(* OpticalPowermeterConfigs *) 
IF Config.OpticalPowermeterConfigs.PM101OpticalPowermeterConfigHs.IsEnabled THEN
	PM101OpticalPowermeterHs.FB_init(FALSE, FALSE, Config := Config.OpticalPowermeterConfigs.PM101OpticalPowermeterConfigHs, 
												   PolarisationConfig := CalibrateConfig.HSPowermeter.PolarisationConfig, 
												   RFactorSettings := CalibrateConfig.HSPowermeter.RFactorSettings,
												   ResponsivityConfig := CalibrateConfig.HSPowermeter.ResponsivityConfig);		
END_IF
IF Config.OpticalPowermeterConfigs.PM101OpticalPowermeterConfigHt.IsEnabled THEN
	PM101OpticalPowermeterHt.FB_init(FALSE, FALSE, Config := Config.OpticalPowermeterConfigs.PM101OpticalPowermeterConfigHt, 
												   PolarisationConfig := CalibrateConfig.HTPowermeter.PolarisationConfig,
												   RFactorSettings := CalibrateConfig.HTPowermeter.RFactorSettings,
												   ResponsivityConfig := CalibrateConfig.HTPowermeter.ResponsivityConfig);
END_IF

(* DistanceSensorConfigs *) 
IF Config.DistanceSensorConfigs.MicroEpsilonDistanceSensorConfig.IsEnabled THEN
	MicroEpsilonDistanceSensor.FB_init(FALSE, FALSE, Config := Config.DistanceSensorConfigs.MicroEpsilonDistanceSensorConfig);	
END_IF

(* MppcConfigs *) 
IF Config.MppcConfigs.C13336MppcConfigWide.IsEnabled THEN
	C13336MppcWide.FB_init(FALSE, FALSE, Config := Config.MppcConfigs.C13336MppcConfigWide);	
END_IF
IF Config.MppcConfigs.C13336MppcConfigNarrow.IsEnabled THEN
	C13336MppcNarrow.FB_init(FALSE, FALSE, Config := Config.MppcConfigs.C13336MppcConfigNarrow);	
END_IF

(* ShutterConfigs *) 
IF Config.ShutterConfigs.Ed12dssShutterConfig.IsEnabled THEN
	Ed12dssShutter.FB_init(FALSE, FALSE, Config := Config.ShutterConfigs.Ed12dssShutterConfig);	
ELSIF Config.ShutterConfigs.SH10PILShutterConfig.IsEnabled THEN
	Sh10pilShutter.FB_init(FALSE, FALSE, Config := Config.ShutterConfigs.SH10PILShutterConfig);	
END_IF

IF Config.IsEnabled THEN
	_logger.Information('Lightspeed devices initialization ended...');
END_IF
END_METHOD

METHOD OpenCloseCycling : BOOL
VAR_INPUT
	Execute : BOOL;
	Count : UINT;
END_VAR
VAR 
END_VAR
IF Execute THEN
	(* timer pour l'enchainement des open/close *)
	(* WaitingTimer.in := TRUE;
	WaitingTimer.PT := T#4S;*)
	WaitingTimer (IN :=TRUE , PT := T#5S,Q=>, ET=> );
	
	(* WaitingTimer.Q is TRUE, PT seconds after IN had a rising edge *)
	IF WaitingTimer.Q THEN
		(* RAZ du timer *)
		WaitingTimer (IN := FALSE);
		(* coupe le motor ON par securité*)
		Chamber.IoLightspeed.OutputDoorslitMotorOn := FALSE;
		(* MAJ du compteur*)
		OpenCloseCyclingCount := Count;
		(* porte ouverte => on demande la fermeture*)
		IF (_CyclingCounterReachSetpoint) THEN
			(* arret du cycling et re init des variables*)
			Chamber.IoLightspeed.OutputDoorslitMotorOn := FALSE;
			_startCycling := FALSE;
			_CyclingCounterReachSetpoint := FALSE;
			_ActivateCyclingMotorOpen := FALSE;
			OpenCloseCycling := FALSE;
			OpenCloseCurrentCounterValue := 0;
			(* to do lever un timeout vers acquisition si not(_CyclingCounterReachSetpoint) => pb d'open/close  *)
		ELSIF Chamber.IoLightspeed.InputDoorslitOpened THEN
			_ActivateCyclingMotorOpen := FALSE;	
		(* porte fermée => on demande l'ouverture *)			
		ELSIF (Chamber.IoLightspeed.InputDoorslitClosed) THEN
			_ActivateCyclingMotorOpen := TRUE;	
		END_IF
	END_IF
END_IF
END_METHOD

METHOD StopCycling : BOOL
VAR_INPUT
	Execute : BOOL;
END_VAR
VAR 
END_VAR
IF Execute THEN
	(* stop du cycling*)
	(* on attend le porte fermée pour arreter le cycling *)
	IF ( NOT (Chamber.IoLightspeed.InputDoorslitOpened) AND Chamber.IoLightspeed.InputDoorslitClosed)  THEN
		(* arret du cycling et re init des variables*)
		(* arret du cycling *)
		_startCycling := FALSE;
		(* coupe le moteur par securité *)
		Chamber.IoLightspeed.OutputDoorslitMotorOn := FALSE;
		(* fin du stop cycling*)
		_stopCycling:= FALSE;
		(* re init du compteur de cycle *)
		_CyclingCounterReachSetpoint := FALSE;
		OpenCloseCurrentCounterValue := 0;
		OpenCloseCyclingCount := 0;
	END_IF
END_IF
END_METHOD

END_FUNCTION_BLOCK

// ---- Service/PMs/PlcModule.TcPOU
FUNCTION_BLOCK PlcModule
VAR_INPUT
END_VAR
VAR_OUTPUT
END_VAR
VAR
	{attribute 'OPC.UA.DA' := '0'}
	_logger : Logger;	
	{attribute 'OPC.UA.DA' := '0'}
	_message : StringBuilder;	
	
	{attribute 'OPC.UA.DA' := '0'}
	message : STRING;
		
	AmsNetIdMsg : STRING(255);
	
	{attribute 'OPC.UA.DA' := '0'}
	_timerRestartAmsNetId : TON;
	{attribute 'OPC.UA.DA' := '0'}
	_restartAmsNetId : BOOL := TRUE;
	{attribute 'OPC.UA.DA' := '0'}
	FbGetAmsNetId : FB_GetLocalAmsNetId;
	{attribute 'OPC.UA.DA' := '0'}
	FbRestart : TC_Restart;
	{attribute 'OPC.UA.DA' := '0'}
	FbReboot : NT_Reboot;	
	{attribute 'OPC.UA.DA' := '0'}
	_execRestart : BOOL;
	{attribute 'OPC.UA.DA' := '0'}
	_execReboot : BOOL;
	
	{attribute 'OPC.UA.DA' := '0'}
	_stateCmd : INT;
	{attribute 'OPC.UA.DA' := '0'}
	_amsNetId : T_AmsNetId;			
	{attribute 'OPC.UA.DA' := '0'}	
	_amsNetIdWasRead : BOOL;
	{attribute 'OPC.UA.DA' := '0'}
	_amsNetIdBadReading : BOOL;
	{attribute 'OPC.UA.DA' := '0'}
	_execAmsNetId : BOOL;
	
	{attribute 'OPC.UA.DA' := '0'}
	_itemScheduler : INT;
	{attribute 'OPC.UA.DA' := '0'}
	_itemRaisedPropertiesBase : INT;	
	
	
	{attribute 'OPC.UA.DA' := '0'}			  		   
	_raisePropertiesBase : BOOL;
	
	{attribute 'OPC.UA.DA' := '0'}
	_pulseGeneratorBase : TON;
END_VAR

IF NOT _amsNetIdWasRead THEN
	GetAmsNetId();
END_IF

IF _amsNetIdWasRead AND NOT _amsNetIdBadReading THEN
	PlcRestart(_execRestart);
	PlcReboot(_execReboot);
END_IF

RaisePropertiesChangedBase(_raisePropertiesBase);

METHOD GetAmsNetId
VAR_INPUT
END_VAR
CASE _stateCmd OF
	0:  FbGetAmsNetId(bExecute := TRUE, tTimeOut := T#2S);
		_stateCmd := 1;
		
	1:	IF(NOT FbGetAmsNetId.bBusy) THEN
			_amsNetId := FbGetAmsNetId.AddrString;			
			 _logger.Information(_message.Reset().Append('AmsNetId=').Append(_amsNetId).ToString());
			FbGetAmsNetId.bExecute := FALSE;				
			_stateCmd := 100;
		END_IF		
		IF FbGetAmsNetId.bError THEN				
			_stateCmd := 10;
		END_IF													 

		// Issue restarts again GetAmsNetId
		_timerRestartAmsNetId(IN := _restartAmsNetId, PT := T#5S);
		IF _timerRestartAmsNetId.Q THEN
			_restartAmsNetId := FALSE;
			_stateCmd := 0;
		END_IF
		
	10: _logger.Error(_message.Reset().Append('AmsNetId errorId=').Append(UDINT_TO_STRING(FbGetAmsNetId.nErrId)).ToString());
		_amsNetIdBadReading := TRUE;
		_stateCmd := 100;	
		 
	100: _amsNetIdWasRead := TRUE;		 
		 _stateCmd := 0;		
END_CASE
END_METHOD

{attribute 'TcRpcEnable' := '1'}
METHOD PROTECTED PlcReboot
VAR_INPUT
	Execute : BOOL;
END_VAR
IF Execute THEN
	_execReboot := TRUE;
	
	FbReboot();	
	CASE _stateCmd OF												
		0:  _logger.Information(_message.Reset().Append('Reboot').ToString());
			_stateCmd := 1;
		
		1:  FbReboot(NETID := _amsNetId, START := TRUE, TMOUT := T#2S, DELAY := 0);
			_stateCmd := 2;
 
		2: IF(NOT FbReboot.Busy) THEN
				FbReboot.START := FALSE;				
				_stateCmd := 100;
			END_IF		        
			IF FbReboot.ERR THEN				
				_stateCmd := 10;
			END_IF	
	
		10: _logger.Error(_message.Reset().Append('Reboot errorId=').
										   Append(UDINT_TO_STRING(FbReboot.ERRID)).ToString());	
			_stateCmd := 100;
			 
		100: _execReboot := FALSE;
			 _stateCmd := 0;		
	END_CASE
END_IF
END_METHOD

{attribute 'TcRpcEnable' := '1'}
METHOD PROTECTED PlcRestart
VAR_INPUT
	Execute : BOOL;
END_VAR
IF Execute THEN	
	_execRestart := TRUE;
	
	FbRestart();	
	CASE _stateCmd OF												
		0:  _logger.Information(_message.Reset().Append('Restart').ToString());
			_stateCmd := 1;
		
		1:  FbRestart(NETID := _amsNetId, RESTART := TRUE, TMOUT := T#2S);
			_stateCmd := 2;
	 
		2: IF(NOT FbRestart.Busy) THEN
				FbRestart.RESTART := FALSE;				
				_stateCmd := 100;
			END_IF		        
			IF FbRestart.ERR THEN				
				_stateCmd := 10;
			END_IF	
	
		10: _logger.Error(_message.Reset().Append('Restart errorId=').
			  							   Append(UDINT_TO_STRING(FbRestart.ERRID)).ToString());	
			_stateCmd := 100;
			 
		100: _execRestart := FALSE;
			 _stateCmd := 0;		
	END_CASE
END_IF
END_METHOD

{attribute 'TcRpcEnable' := '1'}
METHOD RaisePropertiesChangedBase
VAR_INPUT
	Execute : BOOL;
END_VAR
IF Execute THEN		
	_raisePropertiesBase := TRUE;	
	
	IF _pulseGeneratorBase.Q THEN
		_pulseGeneratorBase(IN := FALSE, PT := T#10MS);
		
		CASE _itemRaisedPropertiesBase OF		
			0: AmsNetIdMsg := ' ';
				_itemRaisedPropertiesBase := 1;
			
			1:  AmsNetIdMsg := TO_STRING(_amsNetId);	   
				_itemRaisedPropertiesBase := 10;
				
			10: 
				_logger.Information(_message.Reset().Append('PLC module - RaisePropertiesChangedBase').ToString());
				_raisePropertiesBase := FALSE;
				_itemRaisedPropertiesBase := 0;
		
		END_CASE
	
	ELSE
		_pulseGeneratorBase(IN := TRUE, PT := T#100MS);	
	END_IF
		
END_IF
END_METHOD

END_FUNCTION_BLOCK

// ---- PMShared/Hardware/Devices/Chambers/Lightspeed/LightspeedChamber.TcPOU
{attribute 'OPC.UA.DA' := '1'}
FUNCTION_BLOCK LightspeedChamber EXTENDS ChamberBase
VAR_INPUT
	IoLightspeed : IoLightspeed;	
	IoSafetyLS : IoSafetyLS;
END_VAR
VAR_OUTPUT
	MppcActivate : BOOL;
END_VAR
VAR
	{attribute 'OPC.UA.DA' := '0'}
	_config : LightspeedChamberConfig;	
	
	{attribute 'OPC.UA.DA' := '0'}
	_initDevice : BOOL;
	
	{attribute 'OPC.UA.DA' := '0'}
	_itemInit : INT;
	{attribute 'OPC.UA.DA' := '0'}
	_pulseGeneratorInit : TON;
	
END_VAR

MppcActivate := IoLightspeed.OutputMppcActivate;

// Init device
InitDevice();

METHOD FB_init : BOOL
VAR_INPUT
	bInitRetains : BOOL; // if TRUE, the retain variables are initialized (warm start / cold start)
	bInCopyCode : BOOL;  // if TRUE, the instance afterwards gets moved into the copy code (online change)
	Config : LightspeedChamberConfig;
END_VAR
IF Config.IsEnabled THEN
	_config := Config;	

	SUPER^._chamberConfig.Name := Config.Name;
	SUPER^._chamberConfig.DeviceID := Config.DeviceID;
	SUPER^._chamberConfig.IsEnabled := Config.IsEnabled;
	SUPER^._chamberConfig.LogLevel := Config.LogLevel;
	
	SUPER^.Name := Config.Name;
	SUPER^.DeviceID := Config.DeviceID;
	
	THIS^.Family := DeviceFamily.Chamber;

	THIS^.SetReady();
	_Logger.Information(_message.Reset().Append('Init ').
							Append('{').Append(TO_STRING(THIS^.Family)).Append('} - ').
							Append('{').Append(TO_STRING(THIS^.Name)).Append('} - ').
							Append('Status : ').Append(TO_STRING(THIS^.Status)).
							ToString());										 
END_IF
END_METHOD

METHOD InitDevice
VAR_INPUT
END_VAR
IF NOT _initDevice THEN			
	IF _pulseGeneratorInit.Q THEN
		_pulseGeneratorInit(IN := FALSE, PT := T#10MS);
			
		CASE _itemInit OF
			0:  _itemInit := 1;
				
			1: _logger.Information(_message.Reset().
								Append(_config.Name).
								Append(' - CoolingFans started').ToString());		
								
				IoLightspeed.OutputCoolingFanFrontPanel := TRUE;
				IoLightspeed.OutputCoolingFanBackPanel := TRUE;
				_initDevice := TRUE;
				_itemInit := 0;
		END_CASE
	ELSE
		_pulseGeneratorInit(IN := TRUE, PT := Const.ACTIVE_TIME_COOLING_FAN);	
	END_IF
END_IF
END_METHOD

{attribute 'TcRpcEnable' := '1'}
METHOD MoveSlitDoorPosition
VAR_INPUT
	Execute : BOOL;
	Position : INT;
END_VAR
IF Execute THEN
	_logger.Information(_message.Reset().Append(_config.Name).Append(' - Move slit door position : ').Append(TO_STRING(Position)).ToString());		

END_IF
END_METHOD

METHOD ReadSlitDoorPosition 
VAR_INPUT
END_VAR
VAR
	open : BOOL;
	close : BOOL;
END_VAR
END_METHOD

END_FUNCTION_BLOCK

// ---- PMShared/Hardware/Devices/Chambers/ChamberBase.TcPOU
FUNCTION_BLOCK ABSTRACT ChamberBase EXTENDS TExecution IMPLEMENTS IDevice
VAR_INPUT
	IoChamberBase : IoChamberBase;
END_VAR
VAR_OUTPUT
END_VAR
VAR
	{attribute 'OPC.UA.DA' := '0'}
	_name : STRING;
	{attribute 'OPC.UA.DA' := '0'}
	_deviceID : STRING;				
	{attribute 'OPC.UA.DA' := '0'}
	_family : DeviceFamily := DeviceFamily.Chamber;		
	{attribute 'OPC.UA.DA' := '0'}
	_logger : Logger;
	{attribute 'OPC.UA.DA' := '0'}
	_message : StringBuilder;
	{attribute 'OPC.UA.DA' := '0'}
	_chamberConfig : DeviceConfiguration;
	
	{attribute 'OPC.UA.DA' := '0'}
	InputIsInMaintenanceMode AT %I* : BOOL;
	{attribute 'OPC.UA.DA' := '0'}
	InputIsInRunMode AT %I* : BOOL;
	{attribute 'OPC.UA.DA' := '0'}
	InputArmNotExtended	AT %I* : BOOL;		
	
	{attribute 'OPC.UA.DA' := '0'}
	_lifeTimeCount : UINT;
	{attribute 'OPC.UA.DA' := '0'}
	_notifyIsAlive : BOOL;
	{attribute 'OPC.UA.DA' := '0'}
	_pulseIsAliveGenerator : TON;
	{attribute 'OPC.UA.DA' := '0'}
	_pulseGeneratorBase : TON;
	{attribute 'OPC.UA.DA' := '0'}
	_execPulseGeneratorBase : TON;	
	
	{attribute 'OPC.UA.DA' := '0'}
	_itemSchedulerBase : INT;
	{attribute 'OPC.UA.DA' := '0'}
	_itemExecSchedulerBase : INT;
	{attribute 'OPC.UA.DA' := '0'}
	_itemRaisedPropertiesBase : INT;	
	
	{attribute 'OPC.UA.DA' := '0'}
	_deliverMessagesBase : INT;
		
	{attribute 'OPC.UA.DA' := '0'}
	_armNotExtendedCmd : BOOL;	
	{attribute 'OPC.UA.DA' := '0'}			  		   
	_raisePropertiesBase : BOOL;	 
	
	{attribute 'OPC.UA.DA' := '0'}
	_extendsArm : BOOL;
	
	StateMsg : STRING(255);
	IsAliveMsg : STRING(255);
	IsInMaintenanceMsg : STRING(255);
	ArmNotExtendedMsg : STRING(255);
	EfemSlitDoorOpenPositionMsg : STRING(255);
	IsReadyToLoadUnloadMsg : STRING(255);	

	{attribute 'OPC.UA.DA' := '0'}
	_slitDoorPosition : ESlitDoorPosition;
	{attribute 'OPC.UA.DA' := '0'}
	_slitDoorOpenPosition : BOOL;
	{attribute 'OPC.UA.DA' := '0'}
	_slitDoorClosePosition : BOOL;
	
	{attribute 'OPC.UA.DA' := '0'}
	ioMessage : STRING;
	
	{attribute 'OPC.UA.DA' := '0'}
	_stageIsInLoadingPosition : BOOL;
END_VAR

// Check if it's still alive	
IF _notifyIsAlive THEN
	IsAliveMsg := TO_STRING(_lifeTimeCount);
	_notifyIsAlive := FALSE;
END_IF

IF HardwareGlobalVariables.ChamberState <> State THEN
	HardwareGlobalVariables.ChamberState := State;
	StateMsg := ANY_TO_STRING(State);		
END_IF


CASE _deliverMessagesBase OF		
	EFeedbackMsgChamberBase.IsInMaintenanceMsg :		
		IsInMaintenanceMsg := ioMessage;	
			
	EFeedbackMsgChamberBase.ArmNotExtendedMsg :				
		ArmNotExtendedMsg := ioMessage;	

	EFeedbackMsgChamberBase.EfemSlitDoorOpenPositionMsg :		
		EfemSlitDoorOpenPositionMsg := ioMessage;	
			
	EFeedbackMsgChamberBase.IsReadyToLoadUnloadMsg :				
		IsReadyToLoadUnloadMsg := ioMessage;	
		
END_CASE

RaisePropertiesChangedBase(_raisePropertiesBase);

IF NOT _armNotExtendedCmd AND NOT _raisePropertiesBase THEN
	MessageSchedulerBase();	
END_IF

{attribute 'TcRpcEnable' := '1'}
METHOD PROTECTED ArmExtendEnabled 
VAR_INPUT
	Execute : BOOL;
	ExtendsArm : BOOL;
END_VAR
VAR
END_VAR
IF Execute THEN	
	(*_armNotExtendedCmd := TRUE;	
	
	_extendsArm := ExtendsArm;

	IF _execPulseGeneratorBase.Q THEN
		_execPulseGeneratorBase(IN := FALSE, PT := T#10MS);
			
		CASE _itemExecSchedulerBase OF
			0:  OutputArmExtendEnabled := _extendsArm;
			
				_logger.Information(_message.Reset().Append('ArmExtendEnabled : ').Append(TO_STRING(_extendsArm)).ToString());			   					
				_itemExecSchedulerBase := 1;
			
			1:  _armNotExtendedCmd := FALSE;	
				_itemExecSchedulerBase := 0;		
								
		END_CASE
	ELSE
		_execPulseGeneratorBase(IN := TRUE, PT := T#50MS);	
	END_IF*)
END_IF
END_METHOD

PROPERTY DeviceID : STRING
GET
DeviceID := _deviceID;
END_GET
SET
_deviceID := DeviceID;
END_SET
END_PROPERTY

PROPERTY Family : DeviceFamily
GET
Family := _family;
END_GET
SET
_family := Family;
END_SET
END_PROPERTY

METHOD GetArmNotExtended
VAR_INPUT
END_VAR
_deliverMessagesBase := EFeedbackMsgChamberBase.ArmNotExtendedMsg;
ioMessage := ANY_TO_STRING(NOT InputArmNotExtended);
END_METHOD

METHOD PROTECTED IsAlive
VAR_INPUT
END_VAR
_notifyIsAlive := TRUE;

IF _lifeTimeCount < 5 THEN
	_lifeTimeCount := _lifeTimeCount + 1;
ELSE
	_lifeTimeCount := 1;
END_IF
END_METHOD

METHOD IsInMaintenance 
VAR_INPUT
END_VAR
_deliverMessagesBase := EFeedbackMsgChamberBase.IsInMaintenanceMsg;

IF InputIsInMaintenanceMode AND NOT InputIsInRunMode THEN
	ioMessage := TO_STRING(TRUE);
ELSIF InputIsInMaintenanceMode AND InputIsInRunMode THEN
ioMessage := TO_STRING(FALSE);
ELSE
	ioMessage := TO_STRING(FALSE);
END_IF
END_METHOD

METHOD IsReadyToLoadUnload
VAR_INPUT
END_VAR
_deliverMessagesBase := EFeedbackMsgChamberBase.IsReadyToLoadUnloadMsg;

// Conditions for authorising the arm to enter the chamber
IF IoChamberBase.InputEfemSlitDoorOpen AND StageIsInLoadingPosition THEN	
	IoChamberBase.OutputIsReadyToLoadUnload := TRUE;
ELSE
	IoChamberBase.OutputIsReadyToLoadUnload := FALSE;
END_IF

ioMessage := ANY_TO_STRING(IoChamberBase.OutputIsReadyToLoadUnload);
END_METHOD

METHOD MessageSchedulerBase
VAR_INPUT
END_VAR
IF _pulseGeneratorBase.Q THEN
	_pulseGeneratorBase(IN := FALSE, PT := T#10MS);
		
	CASE _itemSchedulerBase OF			
		0:  _deliverMessagesBase := EFeedbackMsgChamberBase.IsInMaintenanceMsg;
			ioMessage := ' ';
			_itemSchedulerBase := 1;
			
		1:	IsInMaintenance(); 
			_itemSchedulerBase := 2;

		2:  _deliverMessagesBase := EFeedbackMsgChamberBase.ArmNotExtendedMsg;
			ioMessage := ' ';
			_itemSchedulerBase := 3;
			
		3:	GetArmNotExtended(); 
			_itemSchedulerBase := 4;	
			
		4:  _deliverMessagesBase := EFeedbackMsgChamberBase.EfemSlitDoorOpenPositionMsg; 
			ioMessage := ' ';		
			_itemSchedulerBase := 5;
			
		5:	ReadEfemSlitDoorPosition(); 
			_itemSchedulerBase := 6;	
			
		6:	_deliverMessagesBase := EFeedbackMsgChamberBase.IsReadyToLoadUnloadMsg;
			ioMessage := ' ';
		   _itemSchedulerBase := 7;
		   
		7:	IsReadyToLoadUnload(); 
			_itemSchedulerBase := 0;	
		
	END_CASE
ELSE
	_pulseGeneratorBase(IN := TRUE, PT := T#50MS);		
END_IF


IF _pulseIsAliveGenerator.Q THEN
	_pulseIsAliveGenerator(IN := FALSE, PT := T#10MS);
		
	IsAlive();	
ELSE
	_pulseIsAliveGenerator(IN := TRUE, PT := T#1000MS);		
END_IF
END_METHOD

{attribute 'TcRpcEnable' := '1'}
METHOD ABSTRACT MoveSlitDoorPosition
VAR_INPUT
	Execute : BOOL;
	Position : INT;
END_VAR
END_METHOD

PROPERTY Name : STRING
GET
Name := _name;
END_GET
SET
_name := Name;
END_SET
END_PROPERTY

{attribute 'TcRpcEnable' := '1'}
METHOD RaisePropertiesChangedBase
VAR_INPUT
	Execute : BOOL;
END_VAR
IF Execute THEN		
	_raisePropertiesBase := TRUE;	
	
	IF _pulseGeneratorBase.Q THEN
		_pulseGeneratorBase(IN := FALSE, PT := T#10MS);
		
		CASE _itemRaisedPropertiesBase OF		
			0: IsInMaintenanceMsg := ' ';
				_itemRaisedPropertiesBase := 1;
			
			1: ArmNotExtendedMsg := ' ';		   
				_itemRaisedPropertiesBase := 10;
				
			10: 
				_logger.Information(_message.Reset().
								    Append(_chamberConfig.Name).
								    Append(' - RaisePropertiesChangedBase').ToString());
				_raisePropertiesBase := FALSE;
				_itemRaisedPropertiesBase := 0;
		
		END_CASE
	
	ELSE
		_pulseGeneratorBase(IN := TRUE, PT := T#50MS);	
	END_IF
		
END_IF
END_METHOD

METHOD ReadEfemSlitDoorPosition
VAR_INPUT
END_VAR
_deliverMessagesBase := EFeedbackMsgChamberBase.EfemSlitDoorOpenPositionMsg;

ioMessage := ANY_TO_STRING(IoChamberBase.InputEfemSlitDoorOpen);
END_METHOD

METHOD ABSTRACT ReadSlitDoorPosition
VAR_INPUT
END_VAR
END_METHOD

PROPERTY PUBLIC SlitDoorClosePosition : BOOL
GET
SlitDoorClosePosition := _slitDoorClosePosition;
END_GET
SET
_slitDoorClosePosition := SlitDoorClosePosition;
END_SET
END_PROPERTY

PROPERTY PUBLIC SlitDoorOpenPosition : BOOL
GET
SlitDoorOpenPosition := _slitDoorOpenPosition;
END_GET
SET
_slitDoorOpenPosition := SlitDoorOpenPosition;
END_SET
END_PROPERTY

PROPERTY PUBLIC SlitDoorPosition : ESlitDoorPosition
GET
SlitDoorPosition := _slitDoorPosition;
END_GET
SET
_slitDoorPosition := SlitDoorPosition;
END_SET
END_PROPERTY

PROPERTY PUBLIC StageIsInLoadingPosition : bool
GET
StageIsInLoadingPosition := _stageIsInLoadingPosition;
END_GET
SET
_stageIsInLoadingPosition := StageIsInLoadingPosition;
END_SET
END_PROPERTY

END_FUNCTION_BLOCK

// ---- PMShared/Hardware/Devices/AttenuationFilters/Thorlabs/FW212CAttenuationFilter.TcPOU
{attribute 'OPC.UA.DA' := '1'}
FUNCTION_BLOCK FW212CAttenuationFilter EXTENDS AttenuationFilterBase
VAR_INPUT
END_VAR
VAR_OUTPUT
END_VAR
VAR
	{attribute 'OPC.UA.DA' := '0'}
	_config : FW212CAttenuationFilterConfig;
	{attribute 'OPC.UA.DA' := '0'}
	_coeAccess : CoeAccess;
	{attribute 'OPC.UA.DA' := '0'}
	_initConfigSerialCom : BOOL;	
	{attribute 'OPC.UA.DA' := '0'}
	_serialCom  : SerialCom(Prefix :='', Suffix := Const.CARRIAGE_RETURN);
	{attribute 'OPC.UA.DA' := '0'}
	_refSerialCom : REFERENCE TO SerialCom(Prefix :='', Suffix := Const.CARRIAGE_RETURN) := _serialCom;	 
	{attribute 'OPC.UA.DA' := '0'}
	_isReceived : BOOL;
	
	{attribute 'OPC.UA.DA' := '0'}
	_deliverMessages : INT;
	
	CheckConnectionMsg : STRING(255);
	PositionMsg : STRING(255);
	PositionCountMsg : STRING(255);
	IdMsg : STRING(255);
	CustomMsg : STRING(255);
	
	{region 'Commands'}	
		 
	{attribute 'OPC.UA.DA' := '0'}
	_moveAbsPosition	 : BOOL;
	{attribute 'OPC.UA.DA' := '0'}
	_jogBackwardPosition : BOOL;
	{attribute 'OPC.UA.DA' := '0'}
	_jogForwardPosition  : BOOL;
	{attribute 'OPC.UA.DA' := '0'}
	_customCmd : BOOL;
	{attribute 'OPC.UA.DA' := '0'}			  		   
	_raiseProperties : BOOL;
		 
	{attribute 'OPC.UA.DA' := '0'}
	_calibrateCmd : BOOL;
		 				  
	{endregion}
	
	{attribute 'OPC.UA.DA' := '0'}
	_initDevice : BOOL;	
	 
	{attribute 'OPC.UA.DA' := '0'}
	_pos : LREAL;
	{attribute 'OPC.UA.DA' := '0'}
	_cmd : STRING;	
	{attribute 'OPC.UA.DA' := '0'}
	_itemScheduler : INT;		
	{attribute 'OPC.UA.DA' := '0'}
	_pulseGenerator : TON;	
		
	{attribute 'OPC.UA.DA' := '0'}
	tmpMessage : STRING;	
	{attribute 'OPC.UA.DA' := '0'}
	message : STRING;
	{attribute 'OPC.UA.DA' := '0'}
	_length : INT;		 
	{attribute 'OPC.UA.DA' := '0'}
	_findSuffix : INT;
		
	{attribute 'OPC.UA.DA' := '0'}
	_calibrateStartAngle : LREAL;
	{attribute 'OPC.UA.DA' := '0'}
	_calibrateEndAngle : LREAL;
	{attribute 'OPC.UA.DA' := '0'}
	_angleSteps : LREAL;
	{attribute 'OPC.UA.DA' := '0'}
	_numberAverages : UINT;
	{attribute 'OPC.UA.DA' := '0'}
	_itemCalibrateScheduler : INT;
	{attribute 'OPC.UA.DA' := '0'}
	_itemRaisedProperties : INT;	
	
	{attribute 'OPC.UA.DA' := '0'}
	_itemPos : UINT;
	{attribute 'OPC.UA.DA' := '0'}
	_pulseCalibration : TON;	
	
	{region 'Calibrate'}
	
	{attribute 'OPC.UA.DA' := '0'}
	PowerMsg : STRING;
	{endregion}
			 	
	{attribute 'OPC.UA.DA' := '0'}
	_isOpen : BOOL;
	{attribute 'OPC.UA.DA' := '0'}
	_isWriteClose : BOOL;
	{attribute 'OPC.UA.DA' := '0'}
	ValuesCalibrate : ARRAY [0..1000] OF LREAL;
	{attribute 'OPC.UA.DA' := '0'}
	_counter : UINT;
	{attribute 'OPC.UA.DA' := '0'}
	PowerSum : LREAL;
	{attribute 'OPC.UA.DA' := '0'}
	PowerAverage : LREAL;
	
	{attribute 'OPC.UA.DA' := '0'}
	_pulseMoveGenerator : TON;
	{attribute 'OPC.UA.DA' := '0'}
	_itemMove : INT;
END_VAR


IF NOT InitConfigSerialCom THEN	
	ConfigureSerialCom();
ELSIF THIS^.Status = TExecutionState.Ready THEN	
	IF _refSerialCom.ErrorReceiveId = COMERROR_NOERROR THEN
		_refSerialCom(TxBuffer:= HardwareGlobalVariables.TxBufferAttenuation, 
			 	      RxBuffer:= HardwareGlobalVariables.RxBufferAttenuation);
	END_IF	
	
	// Init device
	InitDevice(); 				  
				  
	// Deliver messages
	IF _refSerialCom.IsReceived THEN
		CASE _deliverMessages OF			
			EFeedbackMsgAttenuationFW212C.CheckConnectionMsg :
				CheckConnectionMsg := _refSerialCom.LastReceivedString;	
			EFeedbackMsgAttenuationFW212C.PositionMsg :
				tmpMessage := DELETE(_refSerialCom.LastReceivedString, 6, 1);
				_length := LEN(tmpMessage);
				_findSuffix := FIND(tmpMessage, Const.CARRIAGE_RETURN);
				message := DELETE(tmpMessage, 4, _findSuffix);	
				
				PositionMsg := message;				
			EFeedbackMsgAttenuationFW212C.PositionCountMsg :
				PositionCountMsg := _refSerialCom.LastReceivedString;
			EFeedbackMsgAttenuationFW212C.IdMsg :
				IdMsg := _refSerialCom.LastReceivedString;
			EFeedbackMsgAttenuationFW212C.CustomMsg :
				CustomMsg := _refSerialCom.LastReceivedString;						
		END_CASE
		
		_deliverMessages := 0;
	END_IF						   	
					
	MoveAbsPosition(_moveAbsPosition, _pos);	
	JogBackwardPosition(_jogBackwardPosition);				
	JogForwardPosition(_jogForwardPosition);
	CustomCommand(_customCmd, _cmd);	
	RaisePropertiesChanged(_raiseProperties);

	IF (NOT _moveAbsPosition AND NOT _jogBackwardPosition AND NOT _jogForwardPosition AND NOT _customCmd
		AND NOT _raiseProperties AND _deliverMessages <> EFeedbackMsgAttenuationFW212C.PositionMsg) THEN
		MessageScheduler();
	END_IF	
END_IF

METHOD CheckConnection
VAR_INPUT
END_VAR
VAR
	cmd : STRING := '';
END_VAR
_deliverMessages := EFeedbackMsgAttenuationFW212C.CheckConnectionMsg;	
_serialCom.Send(cmd);
END_METHOD

METHOD ConfigureSerialCom
VAR_INPUT
END_VAR
VAR
END_VAR
IF _coeAccess.CoeOperation.Ready THEN
	_logger.Information(_message.Reset().Append('Start configuration com serial').ToString());
END_IF;	

_coeAccess.CoeOperation.Start();
_coeAccess(SerialCommunication := _config.SerialCommunication);
	
IF _coeAccess.CoeOperation.Done THEN
	_coeAccess.SetDone();	
 
	_Logger.Information(_message.Reset().
							Append('{').Append(TO_STRING(THIS^.Family)).Append('} : ').
							Append(' - Status : ').Append(TO_STRING(_coeAccess.Status)).ToString());	
	InitConfigSerialCom := TRUE;
END_IF
 
IF _coeAccess.CoeOperation.Error THEN	
	_coeAccess.SetError(0);
	
	_Logger.Error(_message.Reset().
							Append('{').Append(TO_STRING(THIS^.Family)).Append('} : ').
							Append(' - Status : ').Append(TO_STRING(_coeAccess.Status)).ToString());
	InitConfigSerialCom := TRUE;
END_IF

THIS^.Status := _coeAccess.Status;
State := _coeAccess.Status;
END_METHOD

{attribute 'TcRpcEnable' := '1'}
METHOD CustomCommand
VAR_INPUT
	Execute : BOOL;
	Cmd : STRING;
END_VAR
IF Execute THEN
	_logger.Information(_message.Reset().
								Append(_config.Name).
								Append(' - Custom : ').
								Append(Cmd).ToString());
	_deliverMessages := EFeedbackMsgAttenuationFW212C.CustomMsg;									
	_serialCom.Send(Cmd);
	
	_customCmd := FALSE;
END_IF
END_METHOD

METHOD FB_init : BOOL
VAR_INPUT
	bInitRetains : BOOL; // if TRUE, the retain variables are initialized (warm start / cold start)
	bInCopyCode : BOOL;  // if TRUE, the instance afterwards gets moved into the copy code (online change)
	Config : FW212CAttenuationFilterConfig;
END_VAR
VAR
END_VAR
IF Config.IsEnabled THEN
	_config := Config;
	
	SUPER^._attenuationFilterConfig.Name := Config.Name;
	SUPER^._attenuationFilterConfig.DeviceID := Config.DeviceID;
	SUPER^._attenuationFilterConfig.IsEnabled := Config.IsEnabled;
	SUPER^._attenuationFilterConfig.LogLevel := Config.LogLevel;
	
	SUPER^.Name := Config.Name;
	SUPER^.DeviceID := Config.DeviceID;	
	THIS^.Family := DeviceFamily.AttenuationFilter;
	
	_Logger.Information(_message.Reset().Append('Init ').
							Append('{').Append(TO_STRING(THIS^.Family)).Append('} - ').
							Append('{').Append(TO_STRING(Config.Name)).Append('}').ToString());																													
END_IF
END_METHOD

(** Returns the model number and firmware version **)
METHOD GetIdentifier
VAR_INPUT
END_VAR
VAR
	cmd : STRING := '*idn?';
END_VAR
_deliverMessages := EFeedbackMsgAttenuationFW212C.IdMsg;
_serialCom.Send(cmd);
END_METHOD

(** Position Query **)
METHOD PROTECTED GetPosition
VAR_INPUT
END_VAR
VAR
	cmd : STRING := 'pos?';
END_VAR
_deliverMessages := EFeedbackMsgAttenuationFW212C.PositionMsg;
_serialCom.Send(cmd);
END_METHOD

(** Returns the wheel type **)
METHOD GetPositionCount
VAR_INPUT
END_VAR
VAR
	cmd : STRING := 'pcount?';
END_VAR
_deliverMessages := EFeedbackMsgAttenuationFW212C.PositionCountMsg;
_serialCom.Send(cmd);
END_METHOD

PROPERTY InitConfigSerialCom : BOOL
GET
InitConfigSerialCom := _initConfigSerialCom;
END_GET
SET
_initConfigSerialCom := InitConfigSerialCom;
END_SET
END_PROPERTY

METHOD InitDevice 
VAR_INPUT
END_VAR
VAR
END_VAR
IF NOT _initDevice THEN	
	_logger.Information(_message.Reset().
								Append(_config.Name).
								Append(' - Init device').ToString());
										
	// TODO : define max count 
	_itemScheduler := 10;
	
	_initDevice := TRUE;	
END_IF
END_METHOD

{attribute 'TcRpcEnable' := '1'}
(** Decrements the filter position by 1 **)
METHOD PROTECTED JogBackwardPosition
VAR_INPUT
	Execute : BOOL;
END_VAR
VAR
	jogBackwardPos : BYTE := 68;
	posArray       : ARRAY[1..3] OF BYTE := [27, 91, jogBackwardPos];	
END_VAR
IF Execute THEN
	_jogBackwardPosition := TRUE;

	IF _pulseMoveGenerator.Q THEN	
		CASE _itemMove OF							
			0:	_logger.Information(_message.Reset().
											Append(_config.Name).
											Append(' - Jog backward position').ToString());
					
				_serialCom.Send3B(posArray);
				
				_itemMove := 1;
				
			1:  GetPosition();
				_itemMove := 10;	
								
			10:  _jogBackwardPosition := FALSE;
				_itemMove := 0;			
		END_CASE			
	ELSE
		_pulseMoveGenerator(IN := TRUE, PT := T#200MS);	
	END_IF	
END_IF
END_METHOD

{attribute 'TcRpcEnable' := '1'}
(** Increments the filter position by 1 **)
METHOD PROTECTED JogForwardPosition
VAR_INPUT
	Execute : BOOL;
END_VAR
VAR
	jogForwardPos : BYTE := 67;
	posArray      : ARRAY[1..3] OF BYTE := [27, 91, jogForwardPos];
END_VAR
IF Execute THEN
	_jogForwardPosition := TRUE;

	IF _pulseMoveGenerator.Q THEN	
		CASE _itemMove OF							
			0:	_logger.Information(_message.Reset().
											Append(_config.Name).
											Append(' - Jog forward position').ToString());
					
				_serialCom.Send3B(posArray);
				
				_itemMove := 1;
				
			1:  GetPosition();
				_itemMove := 10;	
								
			10:  _jogForwardPosition := FALSE;
				_itemMove := 0;			
		END_CASE			
	ELSE
		_pulseMoveGenerator(IN := TRUE, PT := T#200MS);	
	END_IF	
END_IF
END_METHOD

METHOD MessageScheduler
VAR_INPUT
END_VAR
IF _pulseGenerator.Q THEN
	_pulseGenerator(IN := FALSE, PT := T#10MS);
		
	CASE _itemScheduler OF	
		10:	GetPosition();
			_itemScheduler := 0;
			
		1:  GetPositionCount();
			_itemScheduler := 2;
			
		2:  CheckConnection();
			_itemScheduler := 3;

		3:  GetIdentifier();
			_itemScheduler := 0;								
	END_CASE
ELSE
	_pulseGenerator(IN := TRUE, PT := T#100MS);	
END_IF
END_METHOD

{attribute 'TcRpcEnable' := '1'}
(** Absulute moves the wheel to filter position n **)
METHOD PROTECTED MoveAbsPosition 
VAR_INPUT
	Execute : BOOL;
	Position : LREAL;
END_VAR
VAR
	cmd : STRING := 'pos=';
	cmdConcat : STRING(255);
END_VAR
IF Execute THEN
	_moveAbsPosition := TRUE;

	IF _pulseMoveGenerator.Q THEN	
		CASE _itemMove OF							
			0:	_logger.Information(_message.Reset().
											Append(_config.Name).
											Append(' - Move absolute position : ').Append(TO_STRING(Position)).ToString());
					
				cmdConcat := CONCAT(cmd, TO_STRING(LREAL_TO_INT(Position)));
				_serialCom.Send(cmdConcat);
				
				_itemMove := 1;
				
			1:  GetPosition();
				_itemMove := 10;	
								
			10:  _moveAbsPosition := FALSE;
				_itemMove := 0;			
		END_CASE			
	ELSE
		_pulseMoveGenerator(IN := TRUE, PT := T#100MS);	
	END_IF	
END_IF
END_METHOD

{attribute 'TcRpcEnable' := '1'}
METHOD RaisePropertiesChanged
VAR_INPUT
	Execute : BOOL;
END_VAR
IF Execute THEN
	IF THIS^.Status <> TExecutionState.Ready THEN	
		_raiseProperties := FALSE;
		RETURN;
	END_IF	

	_raiseProperties := TRUE;
	
	IF _pulseGenerator.Q THEN
		_pulseGenerator(IN := FALSE, PT := T#10MS);	

		CASE _itemRaisedProperties OF
			0:	PositionMsg := ' ';
				
				_itemRaisedProperties := 10;
			
			10:  GetPosition();
				_itemRaisedProperties := 11;
							
			11:  _logger.Information(_message.Reset().
								Append(_config.Name).
								Append(' - Attenuation RaisePropertiesChanged').ToString());
				_raiseProperties := FALSE;				
				_itemRaisedProperties := 0;
			
		END_CASE
	ELSE
		_pulseGenerator(IN := TRUE, PT := T#100MS);	
	END_IF
END_IF
END_METHOD

END_FUNCTION_BLOCK

// ---- PMShared/Hardware/Devices/AttenuationFilters/AttenuationFilterBase.TcPOU
FUNCTION_BLOCK ABSTRACT AttenuationFilterBase EXTENDS TExecution IMPLEMENTS IDevice
VAR_INPUT
END_VAR
VAR_OUTPUT
END_VAR
VAR
	{attribute 'OPC.UA.DA' := '0'}
	_name : STRING;
	{attribute 'OPC.UA.DA' := '0'}
	_deviceID : STRING;					
	{attribute 'OPC.UA.DA' := '0'}
	_family : DeviceFamily;				
	{attribute 'OPC.UA.DA' := '0'}
	_logger : Logger;
	{attribute 'OPC.UA.DA' := '0'}
	_message : StringBuilder;	
	{attribute 'OPC.UA.DA' := '0'}
	_attenuationFilterConfig : DeviceConfiguration;
END_VAR

PROPERTY DeviceID : STRING
GET
DeviceID := _deviceID;
END_GET
SET
_deviceID := DeviceID;
END_SET
END_PROPERTY

PROPERTY Family : DeviceFamily
GET
Family := _family;
END_GET
SET
_family := Family;
END_SET
END_PROPERTY

METHOD PROTECTED ABSTRACT GetPosition
VAR_INPUT
END_VAR
END_METHOD

METHOD PROTECTED ABSTRACT JogBackwardPosition
VAR_INPUT
	Execute : BOOL;
END_VAR
END_METHOD

METHOD PROTECTED ABSTRACT JogForwardPosition
VAR_INPUT
	Execute : BOOL;
END_VAR
END_METHOD

METHOD PROTECTED ABSTRACT MoveAbsPosition
VAR_INPUT
	Execute : BOOL;
	Position : LREAL;
END_VAR
END_METHOD

PROPERTY Name : STRING
GET
Name := _name;
END_GET
SET
_name := Name;
END_SET
END_PROPERTY

END_FUNCTION_BLOCK

// ---- PMShared/Hardware/Common/Tools/CoeAccess/CoeAccess.TcPOU
FUNCTION_BLOCK CoeAccess EXTENDS TExecution
VAR_INPUT
	SerialCommunication : SerialCommunication;
END_VAR
VAR_OUTPUT
END_VAR
VAR
	_logger : Logger;	
	_message : StringBuilder;
	_coeWrite  : FB_EcCoESdoWrite;
	_coeOperation : TExecution;
	
	_netId     : T_AmsNetId := GlobalConfig.AppConfig.NetIdManagement.FirstPeripheral;
    _slaveAddr : UINT;
	_subIndex  : BYTE;
	_index	   : WORD;
	_bufferLengh : UDINT;
		
	_stateConfig : BYTE := 0;
	_dataSend : UDINT;
	
	item : INT;
END_VAR

SerialCom(_coeOperation.Starting);

IF _coeWrite.bBusy THEN
    _coeOperation.SetBusy();
END_IF

IF _coeWrite.bError THEN
	_coeOperation.SetError(ErrorId := _coeWrite.nErrId);
		
	_logger.Error(_message.Reset().Append('CoE access operation - ErrorId : ').
			 			   		   Append(UDINT_TO_STRING(_coeWrite.nErrId)).ToString());
END_IF 

IF _coeOperation.Busy THEN
    IF NOT _coeWrite.bBusy THEN        
        IF THIS^.Aborted THEN
            _coeOperation.SetAborted();
			_logger.Information(_message.Reset().Append('CoE access operation aborted').ToString());
        ELSIF THIS^.Done THEN             
			_logger.Debug(_message.Reset().Append('CoE access operation done').ToString());
        END_IF
    END_IF
END_IF

METHOD PRIVATE BaudrateValue : UDINT
VAR_INPUT
	value : UDINT;
END_VAR
VAR
	concatValue : STRING;
END_VAR

concatValue := Concat('_', TO_STRING(value));

IF TO_STRING(EBaudrate._9600) = concatValue THEN
	BaudrateValue := ANY_TO_UDINT(EBaudrate._9600);
ELSIF TO_STRING(EBaudrate._19200) = concatValue THEN
	BaudrateValue := ANY_TO_UDINT(EBaudrate._19200);
ELSIF TO_STRING(EBaudrate._38400) = concatValue THEN
	BaudrateValue := ANY_TO_UDINT(EBaudrate._38400);
ELSIF TO_STRING(EBaudrate._57600) = concatValue THEN
	BaudrateValue := ANY_TO_UDINT(EBaudrate._57600);
ELSIF TO_STRING(EBaudrate._115200) = concatValue THEN
	BaudrateValue := ANY_TO_UDINT(EBaudrate._115200);	
ELSE
	_logger.Error(_message.Reset().
						Append('Error serial communication - BaudrateValue : ').
						Append(TO_STRING(value)).ToString());
END_IF;
END_METHOD

PROPERTY BufferLengh : UDINT
GET
BufferLengh := _bufferLengh;
END_GET
SET
_bufferLengh := BufferLengh;
END_SET
END_PROPERTY

PROPERTY CoeOperation : IExecution
GET
CoeOperation := _coeOperation;
END_GET
END_PROPERTY

METHOD PRIVATE DataFrameValue : UDINT
VAR_INPUT
	value : STRING;
END_VAR
VAR
	concatValue : STRING;
END_VAR

concatValue := Concat('_', TO_STRING(value));

IF TO_STRING(EDataFrame._8N1) = concatValue THEN
	DataFrameValue := ANY_TO_UDINT(EDataFrame._8N1);
ELSIF TO_STRING(EDataFrame._8E1) = concatValue THEN
	DataFrameValue := ANY_TO_UDINT(EDataFrame._8E1);
ELSE
	_logger.Error(_message.Reset().
						Append('Error serial communication - DataFrameValue : ').
						Append(value).ToString());	
END_IF;
END_METHOD

PROPERTY Index : WORD
GET
Index := _index;
END_GET
SET
_index := Index;
END_SET
END_PROPERTY

PROPERTY NetId : T_AmsNetId
GET
NetId := _netId;
END_GET
SET
_netId := NetId;
END_SET
END_PROPERTY

METHOD SerialCom
VAR_INPUT
	Execute : BOOL;
END_VAR
VAR
	sIndex : STRING;
	sSubIndex : STRING;
END_VAR
IF item = 0 THEN	

	THIS^.State := TExecutionState.Busy;
	_coeWrite(bExecute := FALSE);	

	CASE _stateConfig OF
	0:	
		// Index
		IF (SerialCommunication.Port = Const.SERIAL_COM_CHANNEL_1) THEN					
			sIndex := CONCAT('16#', GlobalConfig.AppConfig.CanOverEthercatConfig.CoeSerialComSettings.IndexComPort1);						
		ELSIF (SerialCommunication.Port = Const.SERIAL_COM_CHANNEL_2) THEN
			sIndex := CONCAT('16#', GlobalConfig.AppConfig.CanOverEthercatConfig.CoeSerialComSettings.IndexComPort2);			
		ELSE 
			_logger.Error('Error com port');
		END_IF
		
		// Convert String_To_hexa -> Word hexa 
		Index := STRING_TO_WORD(sIndex);
		_logger.Debug(_message.Reset().Append('Index (Dec): ').Append(TO_STRING(Index)).
									   Append(' -> ').Append(sIndex).
									   Append(' (').Append(SerialCommunication.Port).Append(')').ToString());
			
		// SlaveAddr						
		SlaveAddr := SerialCommunication.CanOverEthercat.AdrEthercat;
		_logger.Debug(_message.Reset().Append('SlaveAddr : ').Append(TO_STRING(SlaveAddr)).ToString());
				
		// Baudrate
		sSubIndex := CONCAT('16#', GlobalConfig.AppConfig.CanOverEthercatConfig.CoeSerialComSettings.BaudRate.SubIndex);		
		SubIndex := STRING_TO_BYTE(sSubIndex);		
		BufferLengh := GlobalConfig.AppConfig.CanOverEthercatConfig.CoeSerialComSettings.BaudRate.SizeByte;
		
		_dataSend := BaudrateValue(SerialCommunication.BaudRate);
		_coeWrite.pSrcBuf := ADR(_dataSend);		 
		
		_logger.Debug(_message.Reset().Append('CoeBaudrate (Dec) : ').Append(TO_STRING(_dataSend)).
							           Append(' [SubIndex : ').Append(sSubIndex).Append(']').
									   Append(' - Send baudrate : ').Append(TO_STRING(SerialCommunication.BaudRate)).ToString());		
	1:
		// DataFrame	
		sSubIndex := CONCAT('16#', GlobalConfig.AppConfig.CanOverEthercatConfig.CoeSerialComSettings.DataFrame.SubIndex);	
		SubIndex := STRING_TO_BYTE(sSubIndex);		
		BufferLengh := GlobalConfig.AppConfig.CanOverEthercatConfig.CoeSerialComSettings.DataFrame.SizeByte;
			
		_dataSend := DataFrameValue(SerialCommunication.DataFrame);
		_coeWrite.pSrcBuf := ADR(_dataSend);
	
		_logger.Debug(_message.Reset().Append('DataFrame (Dec) : ').Append(TO_STRING(_dataSend)).
							  		   Append(' [SubIndex : ').Append(sSubIndex).Append(']').
									   Append(' - Send DataFrame : ').Append(SerialCommunication.DataFrame).ToString());
	2:
		// FlowControl RtsCts
		sSubIndex := CONCAT('16#', GlobalConfig.AppConfig.CanOverEthercatConfig.CoeSerialComSettings.EnableRtsCts.SubIndex);	
		SubIndex := STRING_TO_BYTE(sSubIndex);
		BufferLengh := GlobalConfig.AppConfig.CanOverEthercatConfig.CoeSerialComSettings.EnableRtsCts.SizeByte;
		
		IF SerialCommunication.FlowControl = SerialFlowControl.RtsCts THEN
			_dataSend := 1;
		ELSE
			_dataSend := 0;		
		END_IF		
	
		_coeWrite.pSrcBuf := ADR(_dataSend);
		
		_logger.Debug(_message.Reset().Append('FlowControl RtsCts : ').Append(TO_STRING(UDINT_TO_BIT(_dataSend))).
									   Append(' [SubIndex : ').Append(sSubIndex).Append(']').
									   Append(' - Send FlowControl : ').Append(TO_STRING(SerialCommunication.FlowControl)).ToString());
	3:
		// FlowControl Tx
		sSubIndex := CONCAT('16#', GlobalConfig.AppConfig.CanOverEthercatConfig.CoeSerialComSettings.EnableXonXoffTx.SubIndex);	
		SubIndex := STRING_TO_BYTE(sSubIndex);
		BufferLengh := GlobalConfig.AppConfig.CanOverEthercatConfig.CoeSerialComSettings.EnableXonXoffTx.SizeByte;
		
		IF SerialCommunication.FlowControl = SerialFlowControl.XonXoff THEN
			_dataSend := 1;
		ELSE
			_dataSend := 0;		
		END_IF		
	
		_coeWrite.pSrcBuf := ADR(_dataSend);
	
		_logger.Debug(_message.Reset().Append('FlowControl Tx : ').Append(TO_STRING(UDINT_TO_BIT(_dataSend))).
								       Append(' [SubIndex : ').Append(sSubIndex).Append(']').
									   Append(' - Send FlowControl : ').Append(TO_STRING(SerialCommunication.FlowControl)).ToString());
	4:
		// FlowControl Rx
		sSubIndex := CONCAT('16#', GlobalConfig.AppConfig.CanOverEthercatConfig.CoeSerialComSettings.EnableXonXoffRx.SubIndex);	
		SubIndex := STRING_TO_BYTE(sSubIndex);
		BufferLengh := GlobalConfig.AppConfig.CanOverEthercatConfig.CoeSerialComSettings.EnableXonXoffRx.SizeByte; 
		
		IF SerialCommunication.FlowControl = SerialFlowControl.XonXoff THEN
			_dataSend := 1;
		ELSE
			_dataSend := 0;		
		END_IF		
	
		_coeWrite.pSrcBuf := ADR(_dataSend);		
	
		_logger.Debug(_message.Reset().Append('FlowControl Rx : ').Append(TO_STRING(UDINT_TO_BIT(_dataSend))).
									   Append(' [SubIndex : ').Append(sSubIndex).Append(']').
									   Append(' - Send FlowControl : ').Append(TO_STRING(SerialCommunication.FlowControl)).ToString());
	END_CASE
END_IF

CASE item OF 	
0:
	_coeWrite(
	sNetId     := NetId,
	nSlaveAddr := SlaveAddr,
	nSubIndex  := SubIndex, 
	nIndex     := Index,    
	cbBufLen   := BufferLengh,
	bExecute   := TRUE,
	tTimeout   := T#1S
	);	
	item := item + 1;
1: 
    _coeWrite();       
    IF _coeWrite.bError THEN
       item := 10;    	  
    ELSE
    	IF NOT _coeWrite.bBusy THEN
			item := 0;    // Done
			
			IF _stateConfig = 4 THEN					
				_coeOperation.SetDone();
				_stateConfig := 0;
			ELSE
				_stateConfig := _stateConfig + 1;
			END_IF		 			 		 		 		 	 
		END_IF
	END_IF		
10:
	// Error handling
	_logger.Error(_message.Reset().
						Append('Error serial communication - ErrorId : ').
						Append(TO_STRING(_coeWrite.nErrId)).ToString());
	
	_stateConfig := 0;
END_CASE
END_METHOD

PROPERTY SlaveAddr : UINT
GET
SlaveAddr := _slaveAddr;
END_GET
SET
_slaveAddr := SlaveAddr;
END_SET
END_PROPERTY

PROPERTY SubIndex : BYTE
GET
SubIndex := _subIndex;
END_GET
SET
_subIndex := SubIndex;
END_SET
END_PROPERTY

END_FUNCTION_BLOCK

// ---- PMShared/Hardware/Common/Tools/SerialCommunication/SerialCom.TcPOU
FUNCTION_BLOCK SerialCom
VAR_INPUT
END_VAR
VAR_OUTPUT
	LastReceivedString : STRING(255);
	IsReceived         : BOOL;
	ErrorReceiveId	   : ComError_t;
	ErrorSendId		   : ComError_t;
END_VAR
VAR_IN_OUT
	TxBuffer : ComBuffer;
	RxBuffer : ComBuffer;
END_VAR
VAR
	_logger  : Logger;
	_message : StringBuilder;
	_prefix  : STRING;
	_suffix  : STRING;
	
	{region 'Send'}		
	_send		 : SendString;
	_send3B		 : SendByte;
	_send6B 	 : SendByte;
	_send8B 	 : SendByte;
	_send9B 	 : SendByte;
	_send12B 	 : SendByte;
	_send32B 	 : SendByte;
	_sendBusy	 : BOOL;
	_sendErrorId : ComError_t;
	_sendError   : BOOL;
	{endregion}
		 
	{region 'Receive'}		 
	_receive		: ReceiveString255;
	_receivedString : STRING(255);	
    _receiveBusy 	: BOOL;
    _receiveErrorId : ComError_t;
    _receiveTimeout : BOOL;
	{endregion}
		 		 
	length  		: INT;
END_VAR


_receive(
	Prefix:= _prefix,
	Suffix:= _suffix, // Carriage return: '$0D' - Line feel  : '$0A'
	ReceivedString:= _receivedString,
	RXbuffer:= RxBuffer,
	StringReceived=> IsReceived,
	Busy=> _receiveBusy,
	Error=> _receiveErrorId,
	RxTimeout=> _receiveTimeout);
	
IF IsReceived THEN
	LastReceivedString := _receivedString;
	ErrorReceiveId := COMERROR_NOERROR;
END_IF

	
IF _receiveErrorId <> COMERROR_NOERROR AND ErrorReceiveId <> _receiveErrorId THEN
	_logger.Error(_message.Reset().Append('Error receiving data - ErrorId : ').
								   Append(TO_STRING(_receiveErrorId)).ToSTRING());
	ErrorReceiveId := _receiveErrorId;
ELSIF _receiveTimeout THEN
	_logger.Error('Error receive timeout');
END_IF

METHOD FB_init : BOOL
VAR_INPUT
	bInitRetains : BOOL; // if TRUE, the retain variables are initialized (warm start / cold start)
	bInCopyCode : BOOL;  // if TRUE, the instance afterwards gets moved into the copy code (online change)
	Prefix : STRING;
    Suffix : STRING;
END_VAR
_prefix := Prefix;
_suffix := Suffix;
END_METHOD

METHOD Send
VAR_INPUT
	Cmd : STRING;
END_VAR
VAR
	tmpConcat : STRING;
END_VAR
// The warning can be disabled here as the user is aware of the risk that the reference may not be valid by checking its validity
{warning disable C0371}

// Checking the VAR_IN_OUT reference, leave the current method in case of invalid reference
IF NOT __ISVALIDREF(TxBuffer) THEN
     RETURN;
END_IF

tmpConcat := CONCAT(_prefix, Cmd);

_send(SendString:= CONCAT(tmpConcat, _suffix), // Carriage return: '$0D' - Line feel  : '$0A'
			TXbuffer:= TxBuffer,
			Busy=> _sendBusy,
			Error=> _sendErrorId);
	
// The warning may be restored at the end of the access area
{warning restore C0371}
	
IF _sendErrorId <> COMERROR_NOERROR AND ErrorSendId <> _sendErrorId THEN
	_logger.Error(_message.Reset().Append('Error sending data - ErrorId : ').
								   Append(TO_STRING(_sendErrorId)).ToSTRING());									
END_IF			

ErrorSendId := _sendErrorId;
END_METHOD

METHOD Send12B
VAR_INPUT
	PosArray : ARRAY[0..11] OF BYTE;
END_VAR
VAR
	counter : UINT;
END_VAR
// The warning can be disabled here as the user is aware of the risk that the reference may not be valid by checking its validity
{warning disable C0371}

// Checking the VAR_IN_OUT reference, leave the current method in case of invalid reference
IF NOT __ISVALIDREF(TxBuffer) THEN
     RETURN;
END_IF

FOR counter:=0 TO SIZEOF(PosArray) BY 1 DO    	
	_send12B (SendByte:= PosArray[counter], 
			   TXbuffer:= TxBuffer,
			   Busy=> _sendBusy,
			   Error=> _sendErrorID);
			
	IF _send12B.Error <> COMERROR_NOERROR AND ErrorSendId <> _sendErrorId THEN
		_logger.Error(_message.Reset().Append('Error sending data - ErrorId : ').
								 	   Append(TO_STRING(_sendErrorId)).ToSTRING());
	END_IF			
END_FOR;

// The warning may be restored at the end of the access area
{warning restore C0371}

ErrorSendId := _sendErrorId;
END_METHOD

METHOD Send32B
VAR_INPUT
	PosArray : ARRAY[0..31] OF BYTE;
END_VAR
VAR
	counter : UINT;
END_VAR
// The warning can be disabled here as the user is aware of the risk that the reference may not be valid by checking its validity
{warning disable C0371}

// Checking the VAR_IN_OUT reference, leave the current method in case of invalid reference
IF NOT __ISVALIDREF(TxBuffer) THEN
     RETURN;
END_IF

FOR counter:=0 TO SIZEOF(PosArray) BY 1 DO    	
	_send12B (SendByte:= PosArray[counter], 
			   TXbuffer:= TxBuffer,
			   Busy=> _sendBusy,
			   Error=> _sendErrorID);
			
	IF _send32B.Error <> COMERROR_NOERROR AND ErrorSendId <> _sendErrorId THEN
		_logger.Error(_message.Reset().Append('Error sending data - ErrorId : ').
								 	   Append(TO_STRING(_sendErrorId)).ToSTRING());
	END_IF			
END_FOR;

// The warning may be restored at the end of the access area
{warning restore C0371}

ErrorSendId := _sendErrorId;
END_METHOD

METHOD Send3B
VAR_INPUT
	PosArray : ARRAY[0..2] OF BYTE;
END_VAR
VAR
	counter : UINT;
END_VAR
// The warning can be disabled here as the user is aware of the risk that the reference may not be valid by checking its validity
{warning disable C0371}

// Checking the VAR_IN_OUT reference, leave the current method in case of invalid reference
IF NOT __ISVALIDREF(TxBuffer) THEN
     RETURN;
END_IF

FOR counter:=0 TO SIZEOF(PosArray) BY 1 DO    	
	_send3B (SendByte:= posArray[counter], 
			TXbuffer:= TxBuffer,
			Busy=> _sendBusy,
			Error=> _sendErrorID);
			
	IF _send3B.Error <> COMERROR_NOERROR THEN
		_logger.Error(_message.Reset().Append('Error sending data - ErrorId : ').
									   Append(TO_STRING(_sendErrorId)).ToSTRING());
	END_IF			
END_FOR;

// The warning may be restored at the end of the access area
{warning restore C0371}

ErrorSendId := _sendErrorId;
END_METHOD

METHOD Send6B
VAR_INPUT
	PosArray : ARRAY[0..5] OF BYTE;
END_VAR
VAR
	counter : UINT;
END_VAR
// The warning can be disabled here as the user is aware of the risk that the reference may not be valid by checking its validity
{warning disable C0371}

// Checking the VAR_IN_OUT reference, leave the current method in case of invalid reference
IF NOT __ISVALIDREF(TxBuffer) THEN
     RETURN;
END_IF

FOR counter:=0 TO SIZEOF(PosArray) BY 1 DO    	
	_send6B (SendByte:= PosArray[counter], 
			   TXbuffer:= TxBuffer,
			   Busy=> _sendBusy,
			   Error=> _sendErrorID);
			
	IF _send6B.Error <> COMERROR_NOERROR THEN
		_logger.Error(_message.Reset().Append('Error sending data - ErrorId : ').Append(TO_STRING(_sendErrorId)).ToSTRING());
	END_IF			
END_FOR;

// The warning may be restored at the end of the access area
{warning restore C0371}

ErrorSendId := _sendErrorId;
END_METHOD

METHOD Send8B
VAR_INPUT
	PosArray : ARRAY[0..7] OF BYTE;
END_VAR
VAR
	counter : UINT;
END_VAR
// The warning can be disabled here as the user is aware of the risk that the reference may not be valid by checking its validity
{warning disable C0371}

// Checking the VAR_IN_OUT reference, leave the current method in case of invalid reference
IF NOT __ISVALIDREF(TxBuffer) THEN
     RETURN;
END_IF

FOR counter:=0 TO SIZEOF(PosArray) BY 1 DO    	
	_send8B (SendByte:= PosArray[counter], 
			   TXbuffer:= TxBuffer,
			   Busy=> _sendBusy,
			   Error=> _sendErrorID);
			
	IF _send8B.Error <> COMERROR_NOERROR THEN
		_logger.Error(_message.Reset().Append('Error sending data - ErrorId : ').Append(TO_STRING(_sendErrorId)).ToSTRING());
	END_IF			
END_FOR;

// The warning may be restored at the end of the access area
{warning restore C0371}

ErrorSendId := _sendErrorId;
END_METHOD

METHOD Send9B
VAR_INPUT
	PosArray : ARRAY[0..8] OF BYTE;
END_VAR
VAR
	counter : UINT;
END_VAR
// The warning can be disabled here as the user is aware of the risk that the reference may not be valid by checking its validity
{warning disable C0371}

// Checking the VAR_IN_OUT reference, leave the current method in case of invalid reference
IF NOT __ISVALIDREF(TxBuffer) THEN
     RETURN;
END_IF

FOR counter:=0 TO SIZEOF(PosArray) BY 1 DO    	
	_send9B (SendByte:= PosArray[counter], 
			   TXbuffer:= TxBuffer,
			   Busy=> _sendBusy,
			   Error=> _sendErrorID);
			
	IF _send9B.Error <> COMERROR_NOERROR THEN
		_logger.Error(_message.Reset().Append('Error sending data - ErrorId : ').Append(TO_STRING(_sendErrorId)).ToSTRING());
	END_IF			
END_FOR;

// The warning may be restored at the end of the access area
{warning restore C0371}

ErrorSendId := _sendErrorId;
END_METHOD

END_FUNCTION_BLOCK

// ---- PMShared/Hardware/Devices/AttenuationFilters/Thorlabs/ELL14KAttenuationFilter.TcPOU
{attribute 'OPC.UA.DA' := '1'}
FUNCTION_BLOCK ELL14KAttenuationFilter EXTENDS AttenuationFilterBase
VAR_INPUT
END_VAR
VAR_OUTPUT
END_VAR
VAR
	{attribute 'OPC.UA.DA' := '0'}
	_config : ELL14KAttenuationFilterConfig;
	{attribute 'OPC.UA.DA' := '0'}
	_coeAccess : CoeAccess;
	{attribute 'OPC.UA.DA' := '0'}
	_initConfigSerialCom : BOOL;	
	{attribute 'OPC.UA.DA' := '0'}
	_serialCom  : SerialCom(Prefix :='', Suffix := Const.CR_LF);
	{attribute 'OPC.UA.DA' := '0'}
	_refSerialCom : REFERENCE TO SerialCom(Prefix :='', Suffix := Const.CR_LF) := _serialCom;	 
	{attribute 'OPC.UA.DA' := '0'}
	_isReceived : BOOL;
	
	{attribute 'OPC.UA.DA' := '0'}
	_deliverMessages : INT;
	
	PositionMsg : STRING(255);
	IdMsg : STRING(255);
	CustomMsg : STRING(255);
	StateMsg : TExecutionState;
	
	{region 'Commands'}	
	
	{attribute 'OPC.UA.DA' := '0'}
	_homePosition 		: BOOL;
	{attribute 'OPC.UA.DA' := '0'}
	_moveAbsPosition    : BOOL;
	{attribute 'OPC.UA.DA' := '0'}
	_moveRelPosition    : BOOL;	
	{attribute 'OPC.UA.DA' := '0'}
	_jogBackwardPosition : BOOL;
	{attribute 'OPC.UA.DA' := '0'}
	_jogForwardPosition  : BOOL;
	{attribute 'OPC.UA.DA' := '0'}
	_customCmd : BOOL;
	{attribute 'OPC.UA.DA' := '0'}			  		   
	_raiseProperties : BOOL;			 
		 
	{endregion}
	
	{attribute 'OPC.UA.DA' := '0'}
	_initDevice : BOOL;	
	 
	{attribute 'OPC.UA.DA' := '0'}
	_pos : LREAL;
	{attribute 'OPC.UA.DA' := '0'}
	_cmd : STRING;	
	{attribute 'OPC.UA.DA' := '0'}
	_itemScheduler : INT;			
	{attribute 'OPC.UA.DA' := '0'}
	_itemRaisedProperties : INT;	
	{attribute 'OPC.UA.DA' := '0'}
	_pulseGenerator : TON;	
			
	{attribute 'OPC.UA.DA' := '0'}
	tmpMessage : STRING;
	{attribute 'OPC.UA.DA' := '0'}
	message : STRING;
	{attribute 'OPC.UA.DA' := '0'}
	_length : INT;		 
	{attribute 'OPC.UA.DA' := '0'}
	_findSuffix : INT;
			
	{attribute 'OPC.UA.DA' := '0'}
	_calibrateStartAngle : LREAL;
	{attribute 'OPC.UA.DA' := '0'}
	_calibrateEndAngle : LREAL;
	{attribute 'OPC.UA.DA' := '0'}
	_angleSteps : LREAL;
	{attribute 'OPC.UA.DA' := '0'}
	_numberAverages : UINT;
	{attribute 'OPC.UA.DA' := '0'}
	_itemCalibrateScheduler : INT;	
	{attribute 'OPC.UA.DA' := '0'}
	_itemPos : UINT;
	{attribute 'OPC.UA.DA' := '0'}
	_pulseCalibration : TON;
		 
	{attribute 'OPC.UA.DA' := '0'}
	PowerMsg : STRING;
		 
	{attribute 'OPC.UA.DA' := '0'}
	_isOpen : BOOL;
	{attribute 'OPC.UA.DA' := '0'}
	_isWriteClose : BOOL;
	{attribute 'OPC.UA.DA' := '0'}
	ValuesCalibrate : ARRAY [0..1000] OF LREAL;
	{attribute 'OPC.UA.DA' := '0'}
	_counter : UINT;
	{attribute 'OPC.UA.DA' := '0'}
	PowerSum : LREAL;
	{attribute 'OPC.UA.DA' := '0'}
	PowerAverage : LREAL;
		 
	{endregion}
	
	{attribute 'OPC.UA.DA' := '0'}
	_lastSetPositionToPulses : DWORD;

	{attribute 'OPC.UA.DA' := '0'}
	InputPiezoBW AT %I* : DINT;
	{attribute 'OPC.UA.DA' := '0'}
	InputPiezoFW AT %I* : DINT;
	{attribute 'OPC.UA.DA' := '0'}
	_rPosition : LREAL; 

END_VAR


IF NOT InitConfigSerialCom THEN
	ConfigureSerialCom();
ELSIF THIS^.Status = TExecutionState.Ready THEN				
	IF _refSerialCom.ErrorReceiveId = COMERROR_NOERROR THEN
		_refSerialCom(TxBuffer:= HardwareGlobalVariables.TxBufferAttenuation, 
		 	      	  RxBuffer:= HardwareGlobalVariables.RxBufferAttenuation);
	END_IF	
				  
	// Init device
	InitDevice(); 				  
				  
	// Deliver messages
	IF _refSerialCom.IsReceived THEN		
		CASE _deliverMessages OF			
			EFeedbackMsgAttenuationELL14K.PositionMsg :				
				tmpMessage := DELETE(_refSerialCom.LastReceivedString, 3, 1);
				_length := LEN(tmpMessage);
				_findSuffix := FIND(tmpMessage, Const.CR_LF);
				message := DELETE(tmpMessage, 4, _findSuffix);
				
				PositionMsg := ConvertPulsesToDegrees(message);	
				_logger.Information(_message.Reset().Append('ELL14KAttenuationFilter position: ').Append(PositionMsg).ToString());				    			
			EFeedbackMsgAttenuationELL14K.IdMsg :
				IdMsg := _refSerialCom.LastReceivedString;
			EFeedbackMsgAttenuationELL14K.CustomMsg :
				CustomMsg := _refSerialCom.LastReceivedString;						
		END_CASE
	ELSE
		CASE _deliverMessages OF			
			EFeedbackMsgAttenuationELL14K.StateMsg :
				StateMsg := State;				
		END_CASE
	END_IF										   	
	
	HomePosition(_homePosition);	
	MoveAbsPosition(_moveAbsPosition, _pos);
	MoveRelPosition(_moveRelPosition, _pos);	
	JogBackwardPosition(_jogBackwardPosition);				
	JogForwardPosition(_jogForwardPosition);
	CustomCommand(_customCmd, _cmd);	
	RaisePropertiesChanged(_raiseProperties);
	
	IF (NOT _homePosition AND NOT _moveAbsPosition AND NOT _moveRelPosition AND NOT _jogBackwardPosition AND NOT _jogForwardPosition 
		AND NOT _customCmd AND NOT _raiseProperties) THEN
		//MessageScheduler();
	END_IF
END_IF

METHOD ConfigureSerialCom
VAR_INPUT
END_VAR
IF _coeAccess.CoeOperation.Ready THEN
	_logger.Information(_message.Reset().Append('Start configuration com serial').ToString());
END_IF;	

_coeAccess.CoeOperation.Start();
_coeAccess(SerialCommunication := _config.SerialCommunication);
	
IF _coeAccess.CoeOperation.Done THEN
	_coeAccess.SetDone();	
 
	_Logger.Information(_message.Reset().
							Append('{').Append(TO_STRING(THIS^.Family)).Append('} : ').
							Append(' - Status : ').Append(TO_STRING(_coeAccess.Status)).ToString());	
	InitConfigSerialCom := TRUE;
END_IF
 
IF _coeAccess.CoeOperation.Error THEN	
	_coeAccess.SetError(0);
	
	_Logger.Error(_message.Reset().
							Append('{').Append(TO_STRING(THIS^.Family)).Append('} : ').
							Append(' - Status : ').Append(TO_STRING(_coeAccess.Status)).ToString());
	InitConfigSerialCom := TRUE;
END_IF

THIS^.Status := _coeAccess.Status;
State := _coeAccess.Status;
END_METHOD

METHOD ConvertDegreesToPulses : STRING
VAR_INPUT
	AnglePosition : LREAL;
END_VAR
VAR
	NumberPulses : DWORD;
	DegreesToPulses : STRING;
END_VAR
NumberPulses := LREAL_TO_DWORD(AnglePosition * Const.PULSES_PER_DEG);	
DegreesToPulses := DWORD_TO_HEXSTR(NumberPulses, 8, FALSE);

_lastSetPositionToPulses := NumberPulses;
ConvertDegreesToPulses := DWORD_TO_HEXSTR(NumberPulses, 8, FALSE );
END_METHOD

METHOD ConvertPulsesToDegrees : STRING;
VAR_INPUT
	Pulses : STRING;
END_VAR
VAR
	pulsesInHex : STRING; 	
	PulsesToDeg : STRING;
	
	pulsesToDowrd : DWORD;
	InterpolationPulsesToDword : DWORD;
	
	gap : INT;
END_VAR
pulsesInHex := CONCAT('16#', Pulses);
pulsesToDowrd := STRING_TO_DWORD(pulsesInHex);

gap := DWORD_TO_INT(_lastSetPositionToPulses) - DWORD_TO_INT(pulsesToDowrd);
(*_logger.Verbose(_message.Reset().Append('gap=').
									 Append(INT_TO_STRING(gap)).ToString());*)

// Interpolation
IF gap > 0 THEN
	InterpolationPulsesToDword := pulsesToDowrd + 1;
ELSIF gap < 0 THEN
	InterpolationPulsesToDword := pulsesToDowrd - 1;	
ELSE
	InterpolationPulsesToDword := pulsesToDowrd;
END_IF

(*_logger.Verbose(_message.Reset().Append(DWORD_TO_STRING(pulsesToDowrd)).Append(';').
									 Append(DWORD_TO_STRING(InterpolationPulsesToDword)).ToString());*)

_rPosition := DWORD_TO_LREAL(InterpolationPulsesToDword) / Const.PULSES_PER_DEG;
PulsesToDeg := LREAL_TO_FMTSTR(_rPosition, 4, TRUE);
ConvertPulsesToDegrees := PulsesToDeg;
END_METHOD

{attribute 'TcRpcEnable' := '1'}
METHOD CustomCommand
VAR_INPUT
	Execute : BOOL;
	Cmd : STRING;
END_VAR
IF Execute THEN
	_logger.Information(_message.Reset().
								Append(_config.Name).
								Append(' - Custom : ').
								Append(Cmd).ToString());
	_deliverMessages := EFeedbackMsgAttenuationELL14K.CustomMsg;									
	_serialCom.Send(Cmd);
	
	_customCmd := FALSE;
END_IF
END_METHOD

METHOD FB_init : BOOL
VAR_INPUT
	bInitRetains : BOOL; // if TRUE, the retain variables are initialized (warm start / cold start)
	bInCopyCode : BOOL;  // if TRUE, the instance afterwards gets moved into the copy code (online change)
	Config : ELL14KAttenuationFilterConfig;
END_VAR
IF Config.IsEnabled THEN
	_config := Config;
	
	SUPER^._attenuationFilterConfig.Name := Config.Name;
	SUPER^._attenuationFilterConfig.DeviceID := Config.DeviceID;
	SUPER^._attenuationFilterConfig.IsEnabled := Config.IsEnabled;
	SUPER^._attenuationFilterConfig.LogLevel := Config.LogLevel;
	
	SUPER^.Name := Config.Name;
	SUPER^.DeviceID := Config.DeviceID;	
	THIS^.Family := DeviceFamily.AttenuationFilter;
	
	_Logger.Information(_message.Reset().Append('Init ').
							Append('{').Append(TO_STRING(THIS^.Family)).Append('} - ').
							Append('{').Append(TO_STRING(Config.Name)).Append('}').ToString());																													
END_IF
END_METHOD

(** Returns the model number and firmware version **)
METHOD GetIdentifier
VAR_INPUT
END_VAR
VAR
	cmd : STRING := '0i1';
END_VAR
_deliverMessages := EFeedbackMsgAttenuationELL14K.IdMsg;	
_serialCom.Send(cmd);
END_METHOD

(** Position Query **)
METHOD PROTECTED GetPosition
VAR_INPUT
END_VAR
VAR
	cmd : STRING := '0gp';
END_VAR
_deliverMessages := EFeedbackMsgAttenuationELL14K.PositionMsg;	
_serialCom.Send(cmd);
END_METHOD

{attribute 'TcRpcEnable' := '1'}
METHOD HomePosition
VAR_INPUT
	Execute : BOOL;
END_VAR
VAR
	cmd : STRING := '0ho1';
END_VAR
IF Execute THEN
	_logger.Information(_message.Reset().
								Append(_config.Name).
								Append(' - Home position : ').ToString());
	_serialCom.Send(cmd);
	
	_homePosition := FALSE;
END_IF
END_METHOD

PROPERTY InitConfigSerialCom : BOOL
GET
InitConfigSerialCom := _initConfigSerialCom;
END_GET
SET
_initConfigSerialCom := InitConfigSerialCom;
END_SET
END_PROPERTY

METHOD InitDevice
VAR_INPUT
END_VAR
IF NOT _initDevice THEN	
	_logger.Information(_message.Reset().
								Append(_config.Name).
								Append(' - Init device').ToString());	
	_initDevice := TRUE;	
	
	GetPosition();
END_IF
END_METHOD

{attribute 'TcRpcEnable' := '1'}
METHOD PROTECTED JogBackwardPosition
VAR_INPUT
	Execute : BOOL;
END_VAR
VAR
	cmd : STRING := '0bw';
END_VAR
IF Execute THEN
	_logger.Information(_message.Reset().
								Append(_config.Name).
								Append(' - Jog backward position : ').ToString());
	_serialCom.Send(cmd);
	
	_jogBackwardPosition := FALSE;
END_IF
END_METHOD

{attribute 'TcRpcEnable' := '1'}
METHOD PROTECTED JogForwardPosition
VAR_INPUT
	Execute : BOOL;
END_VAR
VAR
	cmd : STRING := '0fw';
END_VAR
IF Execute THEN
	_logger.Information(_message.Reset().
								Append(_config.Name).
								Append(' - Jog forward position : ').ToString());
	_serialCom.Send(cmd);
	
	_jogForwardPosition := FALSE;
END_IF
END_METHOD

METHOD MessageScheduler
VAR_INPUT
END_VAR
IF _pulseGenerator.Q THEN
	_pulseGenerator(IN := FALSE, PT := T#10MS);
	
	GetPosition();
ELSE
	_pulseGenerator(IN := TRUE, PT := T#100MS);		
END_IF
END_METHOD

{attribute 'TcRpcEnable' := '1'}
METHOD PROTECTED MoveAbsPosition 
VAR_INPUT
	Execute : BOOL;
	Position : LREAL;
END_VAR
VAR
	cmd : STRING := '0ma';
END_VAR
IF Execute THEN
	_pos := Position;	
	_logger.Information(_message.Reset().
								Append(_config.Name).
								Append(' - Move absolute position : ').Append(TO_STRING(_pos)).ToString());
		
	_serialCom.Send(CONCAT(cmd, ConvertDegreesToPulses(_pos)));
	_moveAbsPosition := FALSE;
END_IF
END_METHOD

{attribute 'TcRpcEnable' := '1'}
METHOD PROTECTED MoveRelPosition 
VAR_INPUT
	Execute : BOOL;
	AnglePosition : LREAL;
END_VAR
VAR
	cmd : STRING := '0mr';
END_VAR
IF Execute THEN
	_pos := AnglePosition;
	_logger.Information(_message.Reset().
								Append(_config.Name).
								Append(' - Move relative position : ').Append(TO_STRING(_pos)).ToString());
	
	_serialCom.Send(CONCAT(cmd, ConvertDegreesToPulses(_pos)));	
	_moveRelPosition := FALSE;
END_IF
END_METHOD

{attribute 'TcRpcEnable' := '1'}
METHOD RaisePropertiesChanged
VAR_INPUT
	Execute : BOOL;
END_VAR
IF Execute THEN
	IF THIS^.Status <> TExecutionState.Ready THEN	
		_raiseProperties := FALSE;
		RETURN;
	END_IF	

	_raiseProperties := TRUE;
	
	IF _pulseGenerator.Q THEN
		_pulseGenerator(IN := FALSE, PT := T#10MS);	

		CASE _itemRaisedProperties OF
			0:  StateMsg := TExecutionState.Unknown;
				PositionMsg := ' ';
				IdMsg := ' ';
				CustomMsg := ' ';
				
				_itemRaisedProperties := 10;
			
			10:  GetIdentifier();
				_itemRaisedProperties := 11;
				
			11: _deliverMessages := EFeedbackMsgAttenuationELL14K.StateMsg;
				_itemRaisedProperties := 12;
				
			12:  GetPosition();
				_itemRaisedProperties := 13;
			
			13:  _logger.Information(_message.Reset().
								Append(_config.Name).
								Append(' - Attenuation RaisePropertiesChanged').ToString());
				_raiseProperties := FALSE;				
				_itemRaisedProperties := 0;
			
		END_CASE
	ELSE
		_pulseGenerator(IN := TRUE, PT := T#100MS);	
	END_IF
END_IF
END_METHOD

END_FUNCTION_BLOCK

// ---- PMShared/Hardware/Devices/AttenuationFilters/Thorlabs/ELL9AttenuationFilter.TcPOU
{attribute 'OPC.UA.DA' := '1'}
FUNCTION_BLOCK ELL9AttenuationFilter EXTENDS AttenuationFilterBase
VAR_INPUT
END_VAR
VAR_OUTPUT
END_VAR
VAR
	{attribute 'OPC.UA.DA' := '0'}
	_config : ELL9AttenuationFilterConfig;
	{attribute 'OPC.UA.DA' := '0'}
	_coeAccess : CoeAccess;
	{attribute 'OPC.UA.DA' := '0'}
	_initConfigSerialCom : BOOL;	
	{attribute 'OPC.UA.DA' := '0'}
	_serialCom  : SerialCom(Prefix :='', Suffix := Const.CR_LF);
	{attribute 'OPC.UA.DA' := '0'}
	_refSerialCom : REFERENCE TO SerialCom(Prefix :='', Suffix := Const.CR_LF) := _serialCom;	 
	{attribute 'OPC.UA.DA' := '0'}
	_isReceived : BOOL;
	
	{attribute 'OPC.UA.DA' := '0'}
	_deliverMessages : INT;
	
	StateMsg : STRING(255);
	StatusMsg : STRING(255);
	IsAliveMsg : STRING(255);
	PositionMsg : STRING(255);
	IdMsg : STRING(255);
	CustomMsg : STRING(255);
	
	{attribute 'OPC.UA.DA' := '0'}
	ForceStatusMsg : STRING(255) := '00';
	
	{region 'Commands'}	
	
	{attribute 'OPC.UA.DA' := '0'}
	_homePosition 		: BOOL;
	{attribute 'OPC.UA.DA' := '0'}
	_moveAbsPosition    : BOOL;
	{attribute 'OPC.UA.DA' := '0'}
	_jogBackwardPosition : BOOL;
	{attribute 'OPC.UA.DA' := '0'}
	_jogForwardPosition  : BOOL;
	{attribute 'OPC.UA.DA' := '0'}
	_customCmd : BOOL;
	{attribute 'OPC.UA.DA' := '0'}			  		   
	_raiseProperties : BOOL;			 
		 
	{endregion}
	
	{attribute 'OPC.UA.DA' := '0'}
	_initDevice : BOOL;	
	 
	{attribute 'OPC.UA.DA' := '0'}
	_pos : LREAL;
	{attribute 'OPC.UA.DA' := '0'}
	_cmd : STRING;	
	{attribute 'OPC.UA.DA' := '0'}
	_itemScheduler : INT;			
	{attribute 'OPC.UA.DA' := '0'}
	_itemRaisedProperties : INT;	
	{attribute 'OPC.UA.DA' := '0'}
	_itemMove : INT;	
	{attribute 'OPC.UA.DA' := '0'}
	_pulseGenerator : TON;
	{attribute 'OPC.UA.DA' := '0'}
	_pulseStatusGenerator : TON;
	{attribute 'OPC.UA.DA' := '0'}
	_pulseMoveGenerator : TON;	
	{attribute 'OPC.UA.DA' := '0'}
	_pulseIsAliveGenerator : TON;	
			
	{attribute 'OPC.UA.DA' := '0'}
	deviceReplyMessage : STRING;
	{attribute 'OPC.UA.DA' := '0'}
	deviceReplyPosition : STRING := '0PO';
	{attribute 'OPC.UA.DA' := '0'}
	deviceReplyStatus : STRING := '0GS';
	{attribute 'OPC.UA.DA' := '0'}
	tmpMessage : STRING;
	{attribute 'OPC.UA.DA' := '0'}
	message : STRING;
	{attribute 'OPC.UA.DA' := '0'}
	_length : INT;		 
	{attribute 'OPC.UA.DA' := '0'}
	_findSuffix : INT;
			
	{attribute 'OPC.UA.DA' := '0'}
	_calibrateStartAngle : LREAL;
	{attribute 'OPC.UA.DA' := '0'}
	_calibrateEndAngle : LREAL;
	{attribute 'OPC.UA.DA' := '0'}
	_angleSteps : LREAL;
	{attribute 'OPC.UA.DA' := '0'}
	_numberAverages : UINT;
	{attribute 'OPC.UA.DA' := '0'}
	_itemCalibrateScheduler : INT;	
	{attribute 'OPC.UA.DA' := '0'}
	_itemPos : UINT;
	{attribute 'OPC.UA.DA' := '0'}
	_pulseCalibration : TON;
		 
	{attribute 'OPC.UA.DA' := '0'}
	PowerMsg : STRING;
		 
	{attribute 'OPC.UA.DA' := '0'}
	_isOpen : BOOL;
	{attribute 'OPC.UA.DA' := '0'}
	_isWriteClose : BOOL;
	{attribute 'OPC.UA.DA' := '0'}
	ValuesCalibrate : ARRAY [0..1000] OF LREAL;
	{attribute 'OPC.UA.DA' := '0'}
	_counter : UINT;
	{attribute 'OPC.UA.DA' := '0'}
	PowerSum : LREAL;
	{attribute 'OPC.UA.DA' := '0'}
	PowerAverage : LREAL;
		 
	{endregion}
	
	{attribute 'OPC.UA.DA' := '0'}
	_lastSetPositionToPulses : DWORD;
	
	{attribute 'OPC.UA.DA' := '0'}
	posToMM : STRING;
	{attribute 'OPC.UA.DA' := '0'}
	pos : UINT; 
	
	{attribute 'OPC.UA.DA' := '0'}
	codeValue : INT;
	{attribute 'OPC.UA.DA' := '0'}
	_delimeter : STRING := ';';
	{attribute 'OPC.UA.DA' := '0'}
	_firstConcat : STRING;

	{attribute 'OPC.UA.DA' := '0'}
	_lifeTimeCount : UINT;
	{attribute 'OPC.UA.DA' := '0'}
	_notifyIsAlive : BOOL;

END_VAR


IF NOT InitConfigSerialCom THEN
	ConfigureSerialCom();
ELSIF THIS^.Status = TExecutionState.Ready THEN				
	IF _refSerialCom.ErrorReceiveId = COMERROR_NOERROR THEN
		_refSerialCom(TxBuffer:= HardwareGlobalVariables.TxBufferAttenuation, 
		 	      	  RxBuffer:= HardwareGlobalVariables.RxBufferAttenuation);
	END_IF	
				  
	// Init device
	InitDevice(); 				  
				  
	// Check if it's still alive
	IF _notifyIsAlive THEN
		IsAliveMsg := TO_STRING(_lifeTimeCount);
		_notifyIsAlive := FALSE;			
	END_IF
	
	IF _deliverMessages = EFeedbackMsgAttenuationELL9.StatusMsg THEN						
		IF StatusMsg <> ForceStatusMsg THEN
			StatusMsg := ForceStatusMsg;
		END_IF
	END_IF
	
	// Deliver messages
	IF _refSerialCom.IsReceived THEN		
		
		deviceReplyMessage := LEFT(_refSerialCom.LastReceivedString, 3);
		IF deviceReplyMessage = deviceReplyPosition THEN
			_deliverMessages := EFeedbackMsgAttenuationELL9.PositionMsg;
		ELSIF deviceReplyMessage = deviceReplyStatus THEN
			_deliverMessages := EFeedbackMsgAttenuationELL9.StatusMsg;		
		END_IF 
		
		CASE _deliverMessages OF	
			EFeedbackMsgAttenuationELL9.StatusMsg :				
				tmpMessage := DELETE(_refSerialCom.LastReceivedString, 3, 1);
				_length := LEN(tmpMessage);
				_findSuffix := FIND(tmpMessage, Const.CR_LF);
				message := DELETE(tmpMessage, 4, _findSuffix);
				
				IF StatusMsg <> message THEN
					StatusMsg := message;
				END_IF
				
			EFeedbackMsgAttenuationELL9.PositionMsg :				
				tmpMessage := DELETE(_refSerialCom.LastReceivedString, 3, 1);
				_length := LEN(tmpMessage);
				_findSuffix := FIND(tmpMessage, Const.CR_LF);
				message := DELETE(tmpMessage, 4, _findSuffix);
				
				posToMM := DWORD_TO_STRING(STRING_TO_DWORD(CONCAT('16#', message)));
				pos := STRING_TO_UINT(posToMM) / (Const.ELL9_TRAVEL / (Const.ELL9_NUMBER_POS-1));
				
				PositionMsg := UINT_TO_STRING(pos);								
				_deliverMessages := 0;
				
				_logger.Information(_message.Reset().
									Append(_config.Name).
									Append(' - PositionMsg: ').Append(PositionMsg).ToString());
																
			EFeedbackMsgAttenuationELL9.IdMsg :
				IdMsg := _refSerialCom.LastReceivedString;
				_logger.Information(_message.Reset().
									Append(_config.Name).
									Append(' - IdMsg: ').Append(IdMsg).ToString());
			EFeedbackMsgAttenuationELL9.CustomMsg :
				CustomMsg := _refSerialCom.LastReceivedString;
				_logger.Information(_message.Reset().
									Append(_config.Name).
									Append(' - CustomMsg: ').Append(CustomMsg).ToString());	
		END_CASE
	ELSE
		CASE _deliverMessages OF			
			EFeedbackMsgAttenuationELL9.StateMsg :				
				StateMsg := ANY_TO_STRING(State);				
		END_CASE
	END_IF										   	
	
	HomePosition(_homePosition);	
	MoveAbsPosition(_moveAbsPosition, _pos);
	JogBackwardPosition(_jogBackwardPosition);				
	JogForwardPosition(_jogForwardPosition);
	CustomCommand(_customCmd, _cmd);	
	RaisePropertiesChanged(_raiseProperties);
	
	IF (NOT _homePosition AND NOT _moveAbsPosition AND NOT _jogBackwardPosition AND NOT _jogForwardPosition 
		AND NOT _customCmd AND NOT _raiseProperties AND _deliverMessages <> EFeedbackMsgAttenuationELL9.PositionMsg) THEN
		MessageScheduler();
	END_IF
END_IF

METHOD ConfigureSerialCom
VAR_INPUT
END_VAR
IF _coeAccess.CoeOperation.Ready THEN
	_logger.Information(_message.Reset().Append('Start configuration com serial').ToString());
END_IF;	

_coeAccess.CoeOperation.Start();
_coeAccess(SerialCommunication := _config.SerialCommunication);
	
IF _coeAccess.CoeOperation.Done THEN
	_coeAccess.SetDone();	
 
	_Logger.Information(_message.Reset().
							Append('{').Append(TO_STRING(THIS^.Family)).Append('} : ').
							Append(' - Status : ').Append(TO_STRING(_coeAccess.Status)).ToString());	
	InitConfigSerialCom := TRUE;
END_IF
 
IF _coeAccess.CoeOperation.Error THEN	
	_coeAccess.SetError(0);
	
	_Logger.Error(_message.Reset().
							Append('{').Append(TO_STRING(THIS^.Family)).Append('} : ').
							Append(' - Status : ').Append(TO_STRING(_coeAccess.Status)).ToString());
	InitConfigSerialCom := TRUE;
END_IF

THIS^.Status := _coeAccess.Status;
State := _coeAccess.Status;
END_METHOD

{attribute 'TcRpcEnable' := '1'}
METHOD CustomCommand
VAR_INPUT
	Execute : BOOL;
	Cmd : STRING;
END_VAR
IF Execute THEN
	_logger.Information(_message.Reset().
								Append(_config.Name).
								Append(' - Custom : ').
								Append(Cmd).ToString());
	_deliverMessages := EFeedbackMsgAttenuationELL9.CustomMsg;									
	_serialCom.Send(Cmd);
	
	_customCmd := FALSE;
END_IF
END_METHOD

METHOD FB_init : BOOL
VAR_INPUT
	bInitRetains : BOOL; // if TRUE, the retain variables are initialized (warm start / cold start)
	bInCopyCode : BOOL;  // if TRUE, the instance afterwards gets moved into the copy code (online change)
	Config : ELL9AttenuationFilterConfig;
END_VAR
IF Config.IsEnabled THEN
	_config := Config;
	
	SUPER^._attenuationFilterConfig.Name := Config.Name;
	SUPER^._attenuationFilterConfig.DeviceID := Config.DeviceID;
	SUPER^._attenuationFilterConfig.IsEnabled := Config.IsEnabled;
	SUPER^._attenuationFilterConfig.LogLevel := Config.LogLevel;
	
	SUPER^.Name := Config.Name;
	SUPER^.DeviceID := Config.DeviceID;	
	THIS^.Family := DeviceFamily.AttenuationFilter;
	
	_Logger.Information(_message.Reset().Append('Init ').
							Append('{').Append(TO_STRING(THIS^.Family)).Append('} - ').
							Append('{').Append(TO_STRING(Config.Name)).Append('}').ToString());																													
END_IF
END_METHOD

(** Returns the model number and firmware version **)
METHOD GetIdentifier
VAR_INPUT
END_VAR
VAR
	cmd : STRING := '0i1';
END_VAR
_deliverMessages := EFeedbackMsgAttenuationELL9.IdMsg;	
_serialCom.Send(cmd);
END_METHOD

(** Position Query **)
METHOD PROTECTED GetPosition
VAR_INPUT
END_VAR
VAR
	cmd : STRING := '0gp';
END_VAR
_deliverMessages := EFeedbackMsgAttenuationELL9.PositionMsg;	
_serialCom.Send(cmd);
END_METHOD

(** Status Query **)
METHOD GetStatus : STRING
VAR_INPUT
END_VAR
VAR
	cmd : STRING := '0gs';
END_VAR
_deliverMessages := EFeedbackMsgAttenuationELL9.StatusMsg;	
_serialCom.Send(cmd);
END_METHOD

{attribute 'TcRpcEnable' := '1'}
METHOD HomePosition
VAR_INPUT
	Execute : BOOL;
END_VAR
VAR
	cmd : STRING := '0ho0';
	statusCodeBusy: STRING(255) := '9';
END_VAR
IF Execute THEN
	StatusMsg := statusCodeBusy;	
	
	_logger.Information(_message.Reset().
								Append(_config.Name).
								Append(' - Home position : ').ToString());
	_serialCom.Send(cmd);
	
	_homePosition := FALSE;
END_IF
END_METHOD

PROPERTY InitConfigSerialCom : BOOL
GET
InitConfigSerialCom := _initConfigSerialCom;
END_GET
SET
_initConfigSerialCom := InitConfigSerialCom;
END_SET
END_PROPERTY

METHOD InitDevice
VAR_INPUT
END_VAR
IF NOT _initDevice THEN	
	_logger.Information(_message.Reset().
								Append(_config.Name).
								Append(' - Init device').ToString());	
	_initDevice := TRUE;	
	
	GetPosition();
END_IF
END_METHOD

METHOD PROTECTED IsAlive
VAR_INPUT
END_VAR
_notifyIsAlive := TRUE;

IF _lifeTimeCount < 5 THEN
	_lifeTimeCount := _lifeTimeCount + 1;
ELSE
	_lifeTimeCount := 1;
END_IF
END_METHOD

{attribute 'TcRpcEnable' := '1'}
METHOD PROTECTED JogBackwardPosition
VAR_INPUT
	Execute : BOOL;
END_VAR
VAR
	cmd : STRING := '0bw';
END_VAR
IF Execute THEN
	_logger.Information(_message.Reset().
								Append(_config.Name).
								Append(' - Jog backward position : ').ToString());
	_serialCom.Send(cmd);
	
	_jogBackwardPosition := FALSE;
END_IF
END_METHOD

{attribute 'TcRpcEnable' := '1'}
METHOD PROTECTED JogForwardPosition
VAR_INPUT
	Execute : BOOL;
END_VAR
VAR
	cmd : STRING := '0fw';
END_VAR
IF Execute THEN
	_logger.Information(_message.Reset().
								Append(_config.Name).
								Append(' - Jog forward position : ').ToString());
	_serialCom.Send(cmd);
	
	_jogForwardPosition := FALSE;
END_IF
END_METHOD

METHOD MessageScheduler
VAR_INPUT
END_VAR
IF _pulseStatusGenerator.Q THEN
	_pulseStatusGenerator(IN := FALSE, PT := T#10MS);
	
	CASE _itemScheduler OF				
		0:	GetStatus();
			_itemScheduler := 0;
	END_CASE		
ELSE
	_pulseStatusGenerator(IN := TRUE, PT := T#100MS);		
END_IF


IF _pulseIsAliveGenerator.Q THEN
	_pulseIsAliveGenerator(IN := FALSE, PT := T#10MS);
		
	IsAlive();	
ELSE
	_pulseIsAliveGenerator(IN := TRUE, PT := T#1000MS);		
END_IF
END_METHOD

{attribute 'TcRpcEnable' := '1'}
METHOD PROTECTED MoveAbsPosition 
VAR_INPUT
	Execute : BOOL;
	Position : LREAL;
END_VAR
VAR
	posToWord : DWORD;
	posInHexa : STRING;	

	positionInHex : STRING;
	cmd : STRING := '0ma';
	
	statusCodeBusy : STRING := '9'; // Cf API 
END_VAR
IF Execute THEN

	_moveAbsPosition := TRUE;
	_pos := Position;	

	IF _pulseMoveGenerator.Q THEN
		_pulseStatusGenerator(IN := FALSE, PT := T#10MS);
	
		CASE _itemMove OF
			0:	IF Position >= 0 AND Position < Const.ELL9_NUMBER_POS THEN
					ForceStatusMsg := statusCodeBusy;
			
					_itemMove := 1;
				ELSE
					_itemMove := 10;
				END_IF
				
			1:	_logger.Information(_message.Reset().
											Append(_config.Name).
											Append(' - Move absolute position : ').Append(TO_STRING(_pos)).ToString());
					
				posToWord := LREAL_TO_DWORD(Position * (Const.ELL9_TRAVEL / (Const.ELL9_NUMBER_POS-1)));	
				posInHexa := DWORD_TO_HEXSTR(posToWord, 8, FALSE);
					
				_serialCom.Send(CONCAT(cmd, posInHexa));
				
				_itemMove := 2;
				
			2:  GetPosition();
				_itemMove := 10;	
								
			10:  _moveAbsPosition := FALSE;
				_itemMove := 0;
				ForceStatusMsg := '00';
			
		END_CASE			
	ELSE
		_pulseMoveGenerator(IN := TRUE, PT := T#100MS);	
	END_IF

END_IF
END_METHOD

{attribute 'TcRpcEnable' := '1'}
METHOD RaisePropertiesChanged
VAR_INPUT
	Execute : BOOL;
END_VAR
IF Execute THEN
	IF THIS^.Status <> TExecutionState.Ready THEN	
		_raiseProperties := FALSE;
		RETURN;
	END_IF	

	_raiseProperties := TRUE;
	
	IF _pulseGenerator.Q THEN
		_pulseGenerator(IN := FALSE, PT := T#10MS);	

		CASE _itemRaisedProperties OF
			0:  StateMsg := ' ';
				PositionMsg := ' ';
				IdMsg := ' ';
				CustomMsg := ' ';
				
				_itemRaisedProperties := 10;
			
			10:  GetIdentifier();
				_itemRaisedProperties := 11;
				
			11: _deliverMessages := EFeedbackMsgAttenuationELL9.StateMsg;
				_itemRaisedProperties := 12;
				
			12:  GetPosition();
				_itemRaisedProperties := 13;
							
			13:  _logger.Information(_message.Reset().
								Append(_config.Name).
								Append(' - Attenuation RaisePropertiesChanged').ToString());
				_raiseProperties := FALSE;				
				_itemRaisedProperties := 0;
			
		END_CASE
	ELSE
		_pulseGenerator(IN := TRUE, PT := T#100MS);	
	END_IF
END_IF
END_METHOD

END_FUNCTION_BLOCK

// ---- PMShared/Hardware/Devices/AttenuationFilters/Thorlabs/ELL6AttenuationFilter.TcPOU
{attribute 'OPC.UA.DA' := '1'}
FUNCTION_BLOCK ELL6AttenuationFilter EXTENDS AttenuationFilterBase
VAR_INPUT
END_VAR
VAR_OUTPUT
END_VAR
VAR
	{attribute 'OPC.UA.DA' := '0'}
	_config : ELL6AttenuationFilterConfig;
	{attribute 'OPC.UA.DA' := '0'}
	_coeAccess : CoeAccess;
	{attribute 'OPC.UA.DA' := '0'}
	_initConfigSerialCom : BOOL;	
	{attribute 'OPC.UA.DA' := '0'}
	_serialCom  : SerialCom(Prefix :='', Suffix := Const.CR_LF);
	{attribute 'OPC.UA.DA' := '0'}
	_refSerialCom : REFERENCE TO SerialCom(Prefix :='', Suffix := Const.CR_LF) := _serialCom;	 
	{attribute 'OPC.UA.DA' := '0'}
	_isReceived : BOOL;
	
	{attribute 'OPC.UA.DA' := '0'}
	_deliverMessages : INT;
	
	PositionMsg : STRING(255);
	IdMsg : STRING(255);
	CustomMsg : STRING(255);
	StateMsg : TExecutionState;
	
	{region 'Commands'}	
	
	{attribute 'OPC.UA.DA' := '0'}
	_homePosition 		: BOOL;
	{attribute 'OPC.UA.DA' := '0'}
	_moveAbsPosition    : BOOL;
	{attribute 'OPC.UA.DA' := '0'}
	_jogBackwardPosition : BOOL;
	{attribute 'OPC.UA.DA' := '0'}
	_jogForwardPosition  : BOOL;
	{attribute 'OPC.UA.DA' := '0'}
	_customCmd : BOOL;
	{attribute 'OPC.UA.DA' := '0'}			  		   
	_raiseProperties : BOOL;			 
		 
	{endregion}
	
	{attribute 'OPC.UA.DA' := '0'}
	_initDevice : BOOL;	
	 
	{attribute 'OPC.UA.DA' := '0'}
	_pos : LREAL;
	{attribute 'OPC.UA.DA' := '0'}
	_cmd : STRING;	
	{attribute 'OPC.UA.DA' := '0'}
	_itemScheduler : INT;			
	{attribute 'OPC.UA.DA' := '0'}
	_itemRaisedProperties : INT;	
	{attribute 'OPC.UA.DA' := '0'}
	_pulseGenerator : TON;	
			
	{attribute 'OPC.UA.DA' := '0'}
	tmpMessage : STRING;
	{attribute 'OPC.UA.DA' := '0'}
	message : STRING;
	{attribute 'OPC.UA.DA' := '0'}
	_length : INT;		 
	{attribute 'OPC.UA.DA' := '0'}
	_findSuffix : INT;
			
	{attribute 'OPC.UA.DA' := '0'}
	_calibrateStartAngle : LREAL;
	{attribute 'OPC.UA.DA' := '0'}
	_calibrateEndAngle : LREAL;
	{attribute 'OPC.UA.DA' := '0'}
	_angleSteps : LREAL;
	{attribute 'OPC.UA.DA' := '0'}
	_numberAverages : UINT;
	{attribute 'OPC.UA.DA' := '0'}
	_itemCalibrateScheduler : INT;	
	{attribute 'OPC.UA.DA' := '0'}
	_itemPos : UINT;
	{attribute 'OPC.UA.DA' := '0'}
	_pulseCalibration : TON;
		 
	{attribute 'OPC.UA.DA' := '0'}
	PowerMsg : STRING;
		 
	{attribute 'OPC.UA.DA' := '0'}
	_isOpen : BOOL;
	{attribute 'OPC.UA.DA' := '0'}
	_isWriteClose : BOOL;
	{attribute 'OPC.UA.DA' := '0'}
	ValuesCalibrate : ARRAY [0..1000] OF LREAL;
	{attribute 'OPC.UA.DA' := '0'}
	_counter : UINT;
	{attribute 'OPC.UA.DA' := '0'}
	PowerSum : LREAL;
	{attribute 'OPC.UA.DA' := '0'}
	PowerAverage : LREAL;
		 
	{endregion}
	
	{attribute 'OPC.UA.DA' := '0'}
	_lastSetPositionToPulses : DWORD;
	
	{attribute 'OPC.UA.DA' := '0'}
	posToMM : STRING;
	{attribute 'OPC.UA.DA' := '0'}
	pos : UINT; 
	

END_VAR


IF NOT InitConfigSerialCom THEN
	ConfigureSerialCom();
ELSIF THIS^.Status = TExecutionState.Ready THEN				
	IF _refSerialCom.ErrorReceiveId = COMERROR_NOERROR THEN
		_refSerialCom(TxBuffer:= HardwareGlobalVariables.RxBufferSliderAttenuation, 
		 	      	  RxBuffer:= HardwareGlobalVariables.RxBufferSliderAttenuation);
	END_IF	
				  
	// Init device
	InitDevice(); 				  
				  
	// Deliver messages
	IF _refSerialCom.IsReceived THEN		
		CASE _deliverMessages OF			
			EFeedbackMsgAttenuationELL6.PositionMsg :				
				tmpMessage := DELETE(_refSerialCom.LastReceivedString, 3, 1);
				_length := LEN(tmpMessage);
				_findSuffix := FIND(tmpMessage, Const.CR_LF);
				message := DELETE(tmpMessage, 4, _findSuffix);
				
				posToMM := DWORD_TO_STRING(STRING_TO_DWORD(CONCAT('16#', message)));
				pos := STRING_TO_UINT(posToMM) / (Const.ELL6_TRAVEL / (Const.ELL6_NUMBER_POS-1));
				
				PositionMsg := UINT_TO_STRING(pos);			    			
			EFeedbackMsgAttenuationELL6.IdMsg :
				IdMsg := _refSerialCom.LastReceivedString;
			EFeedbackMsgAttenuationELL6.CustomMsg :
				CustomMsg := _refSerialCom.LastReceivedString;	
		END_CASE
	ELSE
		CASE _deliverMessages OF			
			EFeedbackMsgAttenuationELL6.StateMsg :
				StateMsg := State;				
		END_CASE
	END_IF										   	
	
	HomePosition(_homePosition);	
	MoveAbsPosition(_moveAbsPosition, _pos);
	JogBackwardPosition(_jogBackwardPosition);				
	JogForwardPosition(_jogForwardPosition);
	CustomCommand(_customCmd, _cmd);	
	RaisePropertiesChanged(_raiseProperties);
	
	IF (NOT _homePosition AND NOT _moveAbsPosition AND NOT _jogBackwardPosition AND NOT _jogForwardPosition 
		AND NOT _customCmd AND NOT _raiseProperties) THEN
		//MessageScheduler();
	END_IF
END_IF

METHOD ConfigureSerialCom
VAR_INPUT
END_VAR
IF _coeAccess.CoeOperation.Ready THEN
	_logger.Information(_message.Reset().Append('Start configuration com serial').ToString());
END_IF;	

_coeAccess.CoeOperation.Start();
_coeAccess(SerialCommunication := _config.SerialCommunication);
	
IF _coeAccess.CoeOperation.Done THEN
	_coeAccess.SetDone();	
 
	_Logger.Information(_message.Reset().
							Append('{').Append(TO_STRING(THIS^.Family)).Append('} : ').
							Append(' - Status : ').Append(TO_STRING(_coeAccess.Status)).ToString());	
	InitConfigSerialCom := TRUE;
END_IF
 
IF _coeAccess.CoeOperation.Error THEN	
	_coeAccess.SetError(0);
	
	_Logger.Error(_message.Reset().
							Append('{').Append(TO_STRING(THIS^.Family)).Append('} : ').
							Append(' - Status : ').Append(TO_STRING(_coeAccess.Status)).ToString());
	InitConfigSerialCom := TRUE;
END_IF

THIS^.Status := _coeAccess.Status;
State := _coeAccess.Status;
END_METHOD

{attribute 'TcRpcEnable' := '1'}
METHOD CustomCommand
VAR_INPUT
	Execute : BOOL;
	Cmd : STRING;
END_VAR
IF Execute THEN
	_logger.Information(_message.Reset().
								Append(_config.Name).
								Append(' - Custom : ').
								Append(Cmd).ToString());
	_deliverMessages := EFeedbackMsgAttenuationELL6.CustomMsg;									
	_serialCom.Send(Cmd);
	
	_customCmd := FALSE;
END_IF
END_METHOD

METHOD FB_init : BOOL
VAR_INPUT
	bInitRetains : BOOL; // if TRUE, the retain variables are initialized (warm start / cold start)
	bInCopyCode : BOOL;  // if TRUE, the instance afterwards gets moved into the copy code (online change)
	Config : ELL6AttenuationFilterConfig;
END_VAR
IF Config.IsEnabled THEN
	_config := Config;
	
	SUPER^._attenuationFilterConfig.Name := Config.Name;
	SUPER^._attenuationFilterConfig.DeviceID := Config.DeviceID;
	SUPER^._attenuationFilterConfig.IsEnabled := Config.IsEnabled;
	SUPER^._attenuationFilterConfig.LogLevel := Config.LogLevel;
	
	SUPER^.Name := Config.Name;
	SUPER^.DeviceID := Config.DeviceID;	
	THIS^.Family := DeviceFamily.AttenuationFilter;
	
	_Logger.Information(_message.Reset().Append('Init ').
							Append('{').Append(TO_STRING(THIS^.Family)).Append('} - ').
							Append('{').Append(TO_STRING(Config.Name)).Append('}').ToString());																													
END_IF
END_METHOD

(** Returns the model number and firmware version **)
METHOD GetIdentifier
VAR_INPUT
END_VAR
VAR
	cmd : STRING := '0i1';
END_VAR
_deliverMessages := EFeedbackMsgAttenuationELL6.IdMsg;	
_serialCom.Send(cmd);
END_METHOD

(** Position Query **)
METHOD PROTECTED GetPosition
VAR_INPUT
END_VAR
VAR
	cmd : STRING := '0po';
END_VAR
_deliverMessages := EFeedbackMsgAttenuationELL6.PositionMsg;	
_serialCom.Send(cmd);
END_METHOD

{attribute 'TcRpcEnable' := '1'}
METHOD HomePosition
VAR_INPUT
	Execute : BOOL;
END_VAR
VAR
	cmd : STRING := '0ho1';
END_VAR
IF Execute THEN
	_logger.Information(_message.Reset().
								Append(_config.Name).
								Append(' - Home position : ').ToString());
	_serialCom.Send(cmd);
	
	_homePosition := FALSE;
END_IF
END_METHOD

PROPERTY InitConfigSerialCom : BOOL
GET
InitConfigSerialCom := _initConfigSerialCom;
END_GET
SET
_initConfigSerialCom := InitConfigSerialCom;
END_SET
END_PROPERTY

METHOD InitDevice
VAR_INPUT
END_VAR
IF NOT _initDevice THEN	
	_logger.Information(_message.Reset().
								Append(_config.Name).
								Append(' - Init device').ToString());	
	_initDevice := TRUE;		
END_IF
END_METHOD

{attribute 'TcRpcEnable' := '1'}
METHOD PROTECTED JogBackwardPosition
VAR_INPUT
	Execute : BOOL;
END_VAR
VAR
	cmd : STRING := '0bw';
END_VAR
IF Execute THEN
	_logger.Information(_message.Reset().
								Append(_config.Name).
								Append(' - Jog backward position : ').ToString());
	_serialCom.Send(cmd);
	
	_jogBackwardPosition := FALSE;
END_IF
END_METHOD

{attribute 'TcRpcEnable' := '1'}
METHOD PROTECTED JogForwardPosition
VAR_INPUT
	Execute : BOOL;
END_VAR
VAR
	cmd : STRING := '0fw';
END_VAR
IF Execute THEN
	_logger.Information(_message.Reset().
								Append(_config.Name).
								Append(' - Jog forward position : ').ToString());
	_serialCom.Send(cmd);
	
	_jogForwardPosition := FALSE;
END_IF
END_METHOD

METHOD MessageScheduler
VAR_INPUT
END_VAR
IF _pulseGenerator.Q THEN
	_pulseGenerator(IN := FALSE, PT := T#10MS);
	
	GetPosition();
ELSE
	_pulseGenerator(IN := TRUE, PT := T#100MS);		
END_IF
END_METHOD

{attribute 'TcRpcEnable' := '1'}
METHOD PROTECTED MoveAbsPosition 
VAR_INPUT
	Execute : BOOL;
	Position : LREAL;
END_VAR
VAR
	posToWord : DWORD;
	posInHexa : STRING;	

	positionInHex : STRING;
	cmd : STRING := '0ma';
END_VAR
IF Execute THEN
	IF Position >= 0 AND Position < Const.ELL6_NUMBER_POS THEN			
		_pos := Position;	
		_logger.Information(_message.Reset().
									Append(_config.Name).
									Append(' - Move absolute position : ').Append(TO_STRING(_pos)).ToString());
			
		posToWord := LREAL_TO_DWORD(Position * (Const.ELL6_TRAVEL / (Const.ELL6_NUMBER_POS-1)));	
		posInHexa := DWORD_TO_HEXSTR(posToWord, 8, FALSE);
			
		_serialCom.Send(CONCAT(cmd, posInHexa));
	END_IF
	_moveAbsPosition := FALSE;
END_IF
END_METHOD

{attribute 'TcRpcEnable' := '1'}
METHOD RaisePropertiesChanged
VAR_INPUT
	Execute : BOOL;
END_VAR
IF Execute THEN
	IF THIS^.Status <> TExecutionState.Ready THEN	
		_raiseProperties := FALSE;
		RETURN;
	END_IF	

	_raiseProperties := TRUE;
	
	IF _pulseGenerator.Q THEN
		_pulseGenerator(IN := FALSE, PT := T#10MS);	

		CASE _itemRaisedProperties OF
			0:  StateMsg := TExecutionState.Unknown;
				PositionMsg := ' ';
				IdMsg := ' ';
				CustomMsg := ' ';
				
				_itemRaisedProperties := 10;
			
			10:  GetIdentifier();
				_itemRaisedProperties := 11;
				
			11: _deliverMessages := EFeedbackMsgAttenuationELL9.StateMsg;
				_itemRaisedProperties := 12;
				
			12:  GetPosition();
				_itemRaisedProperties := 13;
			
			13:  _logger.Information(_message.Reset().
								Append(_config.Name).
								Append(' - Attenuation RaisePropertiesChanged').ToString());
				_raiseProperties := FALSE;				
				_itemRaisedProperties := 0;
			
		END_CASE
	ELSE
		_pulseGenerator(IN := TRUE, PT := T#100MS);	
	END_IF
END_IF
END_METHOD

END_FUNCTION_BLOCK

// ---- PMShared/Hardware/Devices/AttenuationFilters/Thorlabs/ELL18AttenuationFilter.TcPOU
{attribute 'OPC.UA.DA' := '1'}
FUNCTION_BLOCK ELL18AttenuationFilter EXTENDS AttenuationFilterBase
VAR_INPUT
END_VAR
VAR_OUTPUT
END_VAR
VAR
	{attribute 'OPC.UA.DA' := '0'}
	_config : ELL18AttenuationFilterConfig;
	{attribute 'OPC.UA.DA' := '0'}
	_coeAccess : CoeAccess;
	{attribute 'OPC.UA.DA' := '0'}
	_initConfigSerialCom : BOOL;	
	{attribute 'OPC.UA.DA' := '0'}
	_serialCom  : SerialCom(Prefix :='', Suffix := Const.CR_LF);
	{attribute 'OPC.UA.DA' := '0'}
	_refSerialCom : REFERENCE TO SerialCom(Prefix :='', Suffix := Const.CR_LF) := _serialCom;	 
	{attribute 'OPC.UA.DA' := '0'}
	_isReceived : BOOL;
	
	{attribute 'OPC.UA.DA' := '0'}
	_deliverMessages : INT;
	
	PositionMsg : STRING(255);
	IdMsg : STRING(255);
	CustomMsg : STRING(255);
	StateMsg : TExecutionState;
	
	{region 'Commands'}	
	
	{attribute 'OPC.UA.DA' := '0'}
	_homePosition 		: BOOL;
	{attribute 'OPC.UA.DA' := '0'}
	_moveAbsPosition    : BOOL;
	{attribute 'OPC.UA.DA' := '0'}
	_moveRelPosition    : BOOL;	
	{attribute 'OPC.UA.DA' := '0'}
	_jogBackwardPosition : BOOL;
	{attribute 'OPC.UA.DA' := '0'}
	_jogForwardPosition  : BOOL;
	{attribute 'OPC.UA.DA' := '0'}
	_customCmd : BOOL;
	{attribute 'OPC.UA.DA' := '0'}			  		   
	_raiseProperties : BOOL;			 
		 
	{endregion}
	
	{attribute 'OPC.UA.DA' := '0'}
	_initDevice : BOOL;	
	 
	{attribute 'OPC.UA.DA' := '0'}
	_pos : LREAL;
	{attribute 'OPC.UA.DA' := '0'}
	_cmd : STRING;	
	{attribute 'OPC.UA.DA' := '0'}
	_itemScheduler : INT;			
	{attribute 'OPC.UA.DA' := '0'}
	_itemRaisedProperties : INT;	
	{attribute 'OPC.UA.DA' := '0'}
	_pulseGenerator : TON;	
			
	{attribute 'OPC.UA.DA' := '0'}
	tmpMessage : STRING;
	{attribute 'OPC.UA.DA' := '0'}
	message : STRING;
	{attribute 'OPC.UA.DA' := '0'}
	_length : INT;		 
	{attribute 'OPC.UA.DA' := '0'}
	_findSuffix : INT;
			
	{attribute 'OPC.UA.DA' := '0'}
	_calibrateStartAngle : LREAL;
	{attribute 'OPC.UA.DA' := '0'}
	_calibrateEndAngle : LREAL;
	{attribute 'OPC.UA.DA' := '0'}
	_angleSteps : LREAL;
	{attribute 'OPC.UA.DA' := '0'}
	_numberAverages : UINT;
	{attribute 'OPC.UA.DA' := '0'}
	_itemCalibrateScheduler : INT;	
	{attribute 'OPC.UA.DA' := '0'}
	_itemPos : UINT;
	{attribute 'OPC.UA.DA' := '0'}
	_pulseCalibration : TON;
		 
	{attribute 'OPC.UA.DA' := '0'}
	PowerMsg : STRING;
		 
	{attribute 'OPC.UA.DA' := '0'}
	_isOpen : BOOL;
	{attribute 'OPC.UA.DA' := '0'}
	_isWriteClose : BOOL;
	{attribute 'OPC.UA.DA' := '0'}
	ValuesCalibrate : ARRAY [0..1000] OF LREAL;
	{attribute 'OPC.UA.DA' := '0'}
	_counter : UINT;
	{attribute 'OPC.UA.DA' := '0'}
	PowerSum : LREAL;
	{attribute 'OPC.UA.DA' := '0'}
	PowerAverage : LREAL;
		 
	{endregion}
	
	{attribute 'OPC.UA.DA' := '0'}
	_lastSetPositionToPulses : DWORD;

	{attribute 'OPC.UA.DA' := '0'}
	InputPiezoBW AT %I* : DINT;
	{attribute 'OPC.UA.DA' := '0'}
	InputPiezoFW AT %I* : DINT;
	{attribute 'OPC.UA.DA' := '0'}
	_rPosition : LREAL; 

END_VAR


IF NOT InitConfigSerialCom THEN
	ConfigureSerialCom();
ELSIF THIS^.Status = TExecutionState.Ready THEN				
	IF _refSerialCom.ErrorReceiveId = COMERROR_NOERROR THEN
		_refSerialCom(TxBuffer:= HardwareGlobalVariables.TxBufferRotatingSwitch, 
		 	      	  RxBuffer:= HardwareGlobalVariables.RxBufferRotatingSwitch);
	END_IF	
				  
	// Init device
	InitDevice(); 				  
				  
	// Deliver messages
	IF _refSerialCom.IsReceived THEN		
		CASE _deliverMessages OF			
			EFeedbackMsgAttenuationELL18.PositionMsg :				
				tmpMessage := DELETE(_refSerialCom.LastReceivedString, 3, 1);
				_length := LEN(tmpMessage);
				_findSuffix := FIND(tmpMessage, Const.CR_LF);
				message := DELETE(tmpMessage, 4, _findSuffix);
				
				PositionMsg := ConvertPulsesToDegrees(message);					    			
			EFeedbackMsgAttenuationELL18.IdMsg :
				IdMsg := _refSerialCom.LastReceivedString;
			EFeedbackMsgAttenuationELL14K.CustomMsg :
				CustomMsg := _refSerialCom.LastReceivedString;						
		END_CASE
	ELSE
		CASE _deliverMessages OF			
			EFeedbackMsgAttenuationELL18.StateMsg :
				StateMsg := State;				
		END_CASE
	END_IF										   	
	
	HomePosition(_homePosition);	
	MoveAbsPosition(_moveAbsPosition, _pos);
	MoveRelPosition(_moveRelPosition, _pos);	
	JogBackwardPosition(_jogBackwardPosition);				
	JogForwardPosition(_jogForwardPosition);
	CustomCommand(_customCmd, _cmd);	
	RaisePropertiesChanged(_raiseProperties);
	
	IF (NOT _homePosition AND NOT _moveAbsPosition AND NOT _moveRelPosition AND NOT _jogBackwardPosition AND NOT _jogForwardPosition 
		AND NOT _customCmd AND NOT _raiseProperties) THEN
		//MessageScheduler();
	END_IF
END_IF

METHOD ConfigureSerialCom
VAR_INPUT
END_VAR
IF _coeAccess.CoeOperation.Ready THEN
	_logger.Information(_message.Reset().Append('Start configuration com serial').ToString());
END_IF;	

_coeAccess.CoeOperation.Start();
_coeAccess(SerialCommunication := _config.SerialCommunication);
	
IF _coeAccess.CoeOperation.Done THEN
	_coeAccess.SetDone();	
 
	_Logger.Information(_message.Reset().
							Append('{').Append(TO_STRING(THIS^.Family)).Append('} : ').
							Append(' - Status : ').Append(TO_STRING(_coeAccess.Status)).ToString());	
	InitConfigSerialCom := TRUE;
END_IF
 
IF _coeAccess.CoeOperation.Error THEN	
	_coeAccess.SetError(0);
	
	_Logger.Error(_message.Reset().
							Append('{').Append(TO_STRING(THIS^.Family)).Append('} : ').
							Append(' - Status : ').Append(TO_STRING(_coeAccess.Status)).ToString());
	InitConfigSerialCom := TRUE;
END_IF

THIS^.Status := _coeAccess.Status;
State := _coeAccess.Status;
END_METHOD

METHOD ConvertDegreesToPulses : STRING
VAR_INPUT
	AnglePosition : LREAL;
END_VAR
VAR
	NumberPulses : DWORD;
	DegreesToPulses : STRING;
END_VAR
NumberPulses := LREAL_TO_DWORD(AnglePosition * Const.PULSES_PER_DEG);	
DegreesToPulses := DWORD_TO_HEXSTR(NumberPulses, 8, FALSE);

_lastSetPositionToPulses := NumberPulses;
ConvertDegreesToPulses := DWORD_TO_HEXSTR(NumberPulses, 8, FALSE );
END_METHOD

METHOD ConvertPulsesToDegrees : STRING;
VAR_INPUT
	Pulses : STRING;
END_VAR
VAR
	pulsesInHex : STRING; 	
	PulsesToDeg : STRING;
	
	pulsesToDowrd : DWORD;
	InterpolationPulsesToDword : DWORD;
	
	gap : INT;
END_VAR
pulsesInHex := CONCAT('16#', Pulses);
pulsesToDowrd := STRING_TO_DWORD(pulsesInHex);

gap := DWORD_TO_INT(_lastSetPositionToPulses) - DWORD_TO_INT(pulsesToDowrd);
(*_logger.Verbose(_message.Reset().Append('gap=').
									 Append(INT_TO_STRING(gap)).ToString());*)

// Interpolation
IF gap > 0 THEN
	InterpolationPulsesToDword := pulsesToDowrd + 1;
ELSIF gap < 0 THEN
	InterpolationPulsesToDword := pulsesToDowrd - 1;	
ELSE
	InterpolationPulsesToDword := pulsesToDowrd;
END_IF

(*_logger.Verbose(_message.Reset().Append(DWORD_TO_STRING(pulsesToDowrd)).Append(';').
									 Append(DWORD_TO_STRING(InterpolationPulsesToDword)).ToString());*)

_rPosition := DWORD_TO_LREAL(InterpolationPulsesToDword) / Const.PULSES_PER_DEG;
PulsesToDeg := LREAL_TO_FMTSTR(_rPosition, 4, TRUE);
ConvertPulsesToDegrees := PulsesToDeg;
END_METHOD

{attribute 'TcRpcEnable' := '1'}
METHOD CustomCommand
VAR_INPUT
	Execute : BOOL;
	Cmd : STRING;
END_VAR
IF Execute THEN
	_logger.Information(_message.Reset().
								Append(_config.Name).
								Append(' - Custom : ').
								Append(Cmd).ToString());
	_deliverMessages := EFeedbackMsgAttenuationELL18.CustomMsg;									
	_serialCom.Send(Cmd);
	
	_customCmd := FALSE;
END_IF
END_METHOD

METHOD FB_init : BOOL
VAR_INPUT
	bInitRetains : BOOL; // if TRUE, the retain variables are initialized (warm start / cold start)
	bInCopyCode : BOOL;  // if TRUE, the instance afterwards gets moved into the copy code (online change)
	Config : ELL18AttenuationFilterConfig;
END_VAR
IF Config.IsEnabled THEN
	_config := Config;
	
	SUPER^._attenuationFilterConfig.Name := Config.Name;
	SUPER^._attenuationFilterConfig.DeviceID := Config.DeviceID;
	SUPER^._attenuationFilterConfig.IsEnabled := Config.IsEnabled;
	SUPER^._attenuationFilterConfig.LogLevel := Config.LogLevel;
	
	SUPER^.Name := Config.Name;
	SUPER^.DeviceID := Config.DeviceID;	
	THIS^.Family := DeviceFamily.AttenuationFilter;
	
	_Logger.Information(_message.Reset().Append('Init ').
							Append('{').Append(TO_STRING(THIS^.Family)).Append('} - ').
							Append('{').Append(TO_STRING(Config.Name)).Append('}').ToString());																													
END_IF
END_METHOD

(** Returns the model number and firmware version **)
METHOD GetIdentifier
VAR_INPUT
END_VAR
VAR
	cmd : STRING := '0i1';
END_VAR
_deliverMessages := EFeedbackMsgAttenuationELL18.IdMsg;	
_serialCom.Send(cmd);
END_METHOD

(** Position Query **)
METHOD PROTECTED GetPosition
VAR_INPUT
END_VAR
VAR
	cmd : STRING := '0gp';
END_VAR
_deliverMessages := EFeedbackMsgAttenuationELL18.PositionMsg;	
_serialCom.Send(cmd);
END_METHOD

{attribute 'TcRpcEnable' := '1'}
METHOD HomePosition
VAR_INPUT
	Execute : BOOL;
END_VAR
VAR
	cmd : STRING := '0ho1';
END_VAR
IF Execute THEN
	_logger.Information(_message.Reset().
								Append(_config.Name).
								Append(' - Home position : ').ToString());
	_serialCom.Send(cmd);
	
	_homePosition := FALSE;
END_IF
END_METHOD

PROPERTY InitConfigSerialCom : BOOL
GET
InitConfigSerialCom := _initConfigSerialCom;
END_GET
SET
_initConfigSerialCom := InitConfigSerialCom;
END_SET
END_PROPERTY

METHOD InitDevice
VAR_INPUT
END_VAR
IF NOT _initDevice THEN	
	_logger.Information(_message.Reset().
								Append(_config.Name).
								Append(' - Init device').ToString());	
	_initDevice := TRUE;	
	
	GetPosition();
END_IF
END_METHOD

{attribute 'TcRpcEnable' := '1'}
METHOD PROTECTED JogBackwardPosition
VAR_INPUT
	Execute : BOOL;
END_VAR
VAR
	cmd : STRING := '0bw';
END_VAR
IF Execute THEN
	_logger.Information(_message.Reset().
								Append(_config.Name).
								Append(' - Jog backward position : ').ToString());
	_serialCom.Send(cmd);
	
	_jogBackwardPosition := FALSE;
END_IF
END_METHOD

{attribute 'TcRpcEnable' := '1'}
METHOD PROTECTED JogForwardPosition
VAR_INPUT
	Execute : BOOL;
END_VAR
VAR
	cmd : STRING := '0fw';
END_VAR
IF Execute THEN
	_logger.Information(_message.Reset().
								Append(_config.Name).
								Append(' - Jog forward position : ').ToString());
	_serialCom.Send(cmd);
	
	_jogForwardPosition := FALSE;
END_IF
END_METHOD

METHOD MessageScheduler
VAR_INPUT
END_VAR
IF _pulseGenerator.Q THEN
	_pulseGenerator(IN := FALSE, PT := T#10MS);
	
	GetPosition();
ELSE
	_pulseGenerator(IN := TRUE, PT := T#100MS);		
END_IF
END_METHOD

{attribute 'TcRpcEnable' := '1'}
METHOD PROTECTED MoveAbsPosition 
VAR_INPUT
	Execute : BOOL;
	Position : LREAL;
END_VAR
VAR
	cmd : STRING := '0ma';
END_VAR
IF Execute THEN
	_pos := Position;	
	_logger.Information(_message.Reset().
								Append(_config.Name).
								Append(' - Move absolute position : ').Append(TO_STRING(_pos)).ToString());
		
	_serialCom.Send(CONCAT(cmd, ConvertDegreesToPulses(_pos)));
	_moveAbsPosition := FALSE;
END_IF
END_METHOD

{attribute 'TcRpcEnable' := '1'}
METHOD PROTECTED MoveRelPosition 
VAR_INPUT
	Execute : BOOL;
	AnglePosition : LREAL;
END_VAR
VAR
	cmd : STRING := '0mr';
END_VAR
IF Execute THEN
	_pos := AnglePosition;
	_logger.Information(_message.Reset().
								Append(_config.Name).
								Append(' - Move relative position : ').Append(TO_STRING(_pos)).ToString());
	
	_serialCom.Send(CONCAT(cmd, ConvertDegreesToPulses(_pos)));	
	_moveRelPosition := FALSE;
END_IF
END_METHOD

{attribute 'TcRpcEnable' := '1'}
METHOD RaisePropertiesChanged
VAR_INPUT
	Execute : BOOL;
END_VAR
IF Execute THEN
	IF THIS^.Status <> TExecutionState.Ready THEN	
		_raiseProperties := FALSE;
		RETURN;
	END_IF	

	_raiseProperties := TRUE;
	
	IF _pulseGenerator.Q THEN
		_pulseGenerator(IN := FALSE, PT := T#10MS);	

		CASE _itemRaisedProperties OF
			0:  StateMsg := TExecutionState.Unknown;
				PositionMsg := ' ';
				IdMsg := ' ';
				CustomMsg := ' ';
				
				_itemRaisedProperties := 10;
			
			10:  GetIdentifier();
				_itemRaisedProperties := 11;
				
			11: _deliverMessages := EFeedbackMsgAttenuationELL18.StateMsg;
				_itemRaisedProperties := 12;
				
			12:  GetPosition();
				_itemRaisedProperties := 13;
			
			13:  _logger.Information(_message.Reset().
								Append(_config.Name).
								Append(' - Attenuation RaisePropertiesChanged').ToString());
				_raiseProperties := FALSE;				
				_itemRaisedProperties := 0;
			
		END_CASE
	ELSE
		_pulseGenerator(IN := TRUE, PT := T#100MS);	
	END_IF
END_IF
END_METHOD

END_FUNCTION_BLOCK

// ---- PMShared/Hardware/Devices/PolarisationFilters/Thorlabs/FW212CPolarisationFilter.TcPOU
{attribute 'OPC.UA.DA' := '1'}
FUNCTION_BLOCK FW212CPolarisationFilter EXTENDS PolarisationFilterBase
VAR_INPUT
END_VAR
VAR_OUTPUT
END_VAR
VAR
	{attribute 'OPC.UA.DA' := '0'}
	_config : FW212CPolarisationFilterConfig;
	{attribute 'OPC.UA.DA' := '0'}
	_coeAccess : CoeAccess;
	{attribute 'OPC.UA.DA' := '0'}
	_initConfigSerialCom : BOOL;
	{attribute 'OPC.UA.DA' := '0'}
	_serialCom  : SerialCom(Prefix :='', Suffix := Const.CARRIAGE_RETURN);
	{attribute 'OPC.UA.DA' := '0'}	
	_refSerialCom : REFERENCE TO SerialCom(Prefix :='', Suffix := Const.CARRIAGE_RETURN) := _serialCom; 
	{attribute 'OPC.UA.DA' := '0'}
	_isReceived : BOOL;
	
	{attribute 'OPC.UA.DA' := '0'}
	_deliverMessages : INT;
	
